Yaskawa INFORM job: SKRZYNIA_5440_0_STOPNI_2OBR.JBI

/JOB
//NAME SKRZYNIA_5440_0_STOPNI_2OBR
///FOLDERNAME 02-SKRZYNIE_JOBS
//POS
///NPOS 734,734,0,54,0,0
///TOOL 0
///POSTYPE PULSE
///PULSE
C00000=1055,-24125,84372,288,19725,204
C00001=0,-15438,65714,0,-68532,0
C00002=4718,-16587,59952,3396,-65485,-935
C00003=32997,-21499,42555,27623,-61436,21376
C00004=31759,-20688,42932,26837,-60850,21559
C00005=28987,-21156,42712,24818,-60442,22222
C00006=33447,-21964,42352,27886,-61721,21330
C00007=37687,-23357,41794,30651,-63289,20620
C00008=38979,-19018,48057,32961,-64962,20678
C00009=37261,-18075,48526,31902,-64209,20901
C00010=35830,-17198,48994,31015,-63571,21092
C00011=34080,-17614,48768,29780,-63290,21485
C00012=37261,-18075,48526,31902,-64209,20901
C00013=47373,-21912,40596,41149,-66086,26950
C00014=4718,-16587,59952,3396,-65485,-935
C00015=32997,-21499,42555,27623,-61436,21376
C00016=31759,-20688,42932,26837,-60850,21559
C00017=28987,-21156,42712,24818,-60442,22222
C00018=33447,-21964,42352,27886,-61721,21330
C00019=37687,-23357,41794,30651,-63289,20620
C00020=38979,-19018,48057,32961,-64962,20678
C00021=37261,-18075,48526,31902,-64209,20901
C00022=35830,-17198,48994,31015,-63571,21092
C00023=34080,-17614,48768,29780,-63290,21485
C00024=37261,-18075,48526,31902,-64209,20901
C00025=47373,-21912,40596,41149,-66086,26950
C00026=45033,-20851,41104,39798,-65001,27223
C00027=42790,-19693,41704,38494,-63946,27495
C00028=41070,-20182,41442,37324,-63566,27891
C00029=45033,-20851,41104,39798,-65001,27223
C00030=45033,-20851,41104,39798,-65001,27223
C00031=59624,-29540,14278,64846,-60867,16042
C00032=57357,-28542,14780,63940,-59509,16120
C00033=56188,-29140,14476,63237,-58995,16387
C00034=59588,-29370,14363,64862,-60819,16012
C00035=62924,-29779,15793,65870,-63073,16252
C00036=59724,-28781,16276,64511,-61238,16415
C00037=57764,-27936,16704,63709,-60078,16488
C00038=56408,-28589,16373,62897,-59486,16787
C00039=59724,-28781,16276,64511,-61238,16415
C00040=59800,-47064,-28857,95901,-51687,-331
C00041=35771,-53551,-30995,85975,-27014,914
C00042=34295,-52413,-30674,86854,-26051,280
C00043=32024,-52970,-30833,85668,-24589,638
C00044=35771,-53551,-30995,85975,-27014,914
C00045=87562,-48087,-13810,78020,-75252,11220
C00046=10104,-46603,4759,11228,-37390,-5046
C00047=0,-52280,40443,0,6876,0
C00048=1529,-42140,58025,-5964,2417,3265
C00049=49472,-39353,6917,53118,-50908,20251
C00050=45058,-39356,3832,51653,-47640,20099
C00051=42883,-38319,4163,50577,-46309,20295
C00052=40255,-38926,3967,48502,-45334,21060
C00053=46774,-39679,3737,52663,-48537,19827
C00054=48708,-40455,3517,53615,-49689,19657
C00055=43798,-39237,3871,50850,-47027,20335
C00056=41951,-38324,4161,49930,-45891,20507
C00057=39836,-38844,3994,48234,-45126,21137
C00058=48489,-40338,3551,53521,-49551,19665
C00059=48489,-40338,3551,53521,-49551,19665
C00060=44432,-39026,3936,51363,-47247,20139
C00061=42487,-38069,4248,50403,-46050,20315
C00062=39061,-38795,4009,47695,-44769,21310
C00063=44432,-39026,3936,51363,-47247,20139
C00064=57930,-43229,1921,58550,-54632,18533
C00065=40247,-55452,-40505,109199,-33003,-7808
C00066=33946,-52082,-43455,125156,-33578,-16149
C00067=32704,-50650,-42908,126591,-33384,-17037
C00068=30549,-51326,-43170,127422,-32071,-17630
C00069=37275,-55997,-51641,126340,-37028,-16651
C00070=64697,-70559,-57820,113226,-48939,-6101
C00071=1817,-44984,2816,-3462,-45659,1296
C00072=1148,-56354,34370,-22,3827,-10
C00073=0,-52280,40443,0,6876,0
C00074=0,-49898,44897,0,-65513,0
C00075=48645,-40151,10421,50724,-47615,19638
C00076=35184,-37395,11059,41539,-41116,22069
C00077=33403,-36378,11356,40435,-40041,22314
C00078=30649,-36829,11220,37805,-39247,23256
C00079=35184,-37395,11059,41539,-41116,22069
C00080=36291,-43239,-398,48566,-36532,18743
C00081=34674,-42363,-182,47694,-35492,18907
C00082=33151,-41445,67,46884,-34487,19058
C00083=30501,-41913,-62,44164,-33547,20068
C00084=34674,-42363,-182,47694,-35492,18907
C00085=54016,-42729,8218,55932,-50472,20462
C00086=-31499,-58302,-23356,15027,12889,-13082
C00087=-52768,-43016,-26078,18373,38595,-18774
C00088=-89470,-32103,-32973,29905,69139,-31512
C00089=-68838,-26884,-24872,16972,64732,-23076
C00090=-53036,-11528,-12218,12363,64665,-17409
C00091=-51536,-9474,-10276,11905,64649,-16876
C00092=-51739,-9114,-7787,12104,63269,-17104
C00093=-53036,-11528,-12218,12363,64665,-17409
C00094=-17541,-26226,-24397,927,59032,-5038
C00095=-17541,-26226,-24397,927,59032,-5038
C00096=-16950,-23991,-22741,715,59568,-4818
C00097=-17036,-23563,-20101,755,58071,-4857
C00098=-17541,-26226,-24397,927,59032,-5038
C00099=34102,-23192,-21614,-15638,64271,13209
C00100=33423,-21885,-20599,-15423,64418,12942
C00101=32426,-19856,-18975,-15106,64629,12551
C00102=32578,-19611,-17013,-15290,63535,12762
C00103=33423,-21885,-20599,-15423,64418,12942
C00104=59339,-6070,-6417,-20979,72191,20891
C00105=59339,-6070,-6417,-20979,72191,20891
C00106=57897,-4256,-4562,-20702,71913,20431
C00107=58108,-3992,-2506,-20878,70835,20713
C00108=59339,-6070,-6417,-20979,72191,20891
C00109=42744,-35904,-30225,-18322,62562,16651
C00110=-53036,-11528,-12218,12363,64665,-17409
C00111=-77982,-26538,-29134,27151,66629,-27745
C00112=-70983,-8594,-1966,26503,59809,-49670
C00113=-80152,19776,40785,37351,72704,-50428
C00114=-79984,20154,42529,37516,71911,-50638
C00115=-79233,18397,40079,37458,71885,-50340
C00116=-79984,20154,42529,37516,71911,-50638
C00117=-73519,23289,38838,28890,77081,-45618
C00118=-73519,24511,42682,29072,75582,-46027
C00119=-73519,23289,38838,28890,77081,-45618
C00120=-88897,15706,42282,50101,71325,-56974
C00121=-88897,15706,42282,50101,71325,-56974
C00122=-87612,12343,37838,50071,70996,-56519
C00123=-85283,14202,40272,50301,69633,-56165
C00124=-87338,12550,38107,50098,70839,-56476
C00125=-84952,-1789,13569,34660,47724,-58955
C00126=-67641,-1674,11109,10330,44856,-44725
C00127=-66443,961,13975,9688,44721,-44210
C00128=-67641,-1674,11109,10330,44856,-44725
C00129=-67641,-376,15347,10694,42950,-44967
C00130=-67641,-1674,11109,10330,44856,-44725
C00131=-79040,417,20398,15965,28992,-57786
C00132=-76655,5212,30978,15501,25024,-57306
C00133=-76655,6949,35816,16758,23084,-57955
C00134=-76655,5212,30978,15501,25024,-57306
C00135=-74761,6919,33010,13466,24593,-56049
C00136=-80460,-2874,12270,15804,32253,-57809
C00137=-61258,-29124,-13156,26560,43617,-22150
C00138=-30420,-40507,-29240,27153,53235,15188
C00139=-18589,-38725,-21450,23338,47896,18931
C00140=-17722,-35233,-16455,23322,46926,19051
C00141=-17722,-33749,-12435,23948,45421,18620
C00142=-17722,-33892,-12819,23887,45564,18661
C00143=-16677,-31133,-11209,23138,46167,19311
C00144=-17819,-35820,-17540,23246,47228,19090
C00145=-74104,-11494,-6266,31916,75042,4269
C00146=-71226,-7329,2631,32115,71468,4273
C00147=-71226,-6504,5446,32343,70365,3922
C00148=-71226,-6611,5086,32313,70505,3967
C00149=-68386,-4058,7675,32040,69573,4789
C00150=-73314,-9412,-353,32206,72648,3829
C00151=51751,-31069,-22965,-10739,49070,48663
C00152=49028,-23852,-11575,-9841,46366,47823
C00153=49028,-23004,-8935,-10039,45204,47956
C00154=49028,-23118,-9286,-10013,45357,47939
C00155=47000,-20813,-7527,-8928,45644,47024
C00156=50476,-26208,-15307,-10408,47325,48332
C00157=90602,-5375,6902,-38786,69848,59444
C00158=83174,19950,50269,-44999,67580,58220
C00159=82362,17902,47383,-44926,67511,57879
C00160=83515,19072,48341,-44798,68200,58056
C00161=78091,19382,40247,-36371,72286,52960
C00162=78091,20664,44011,-36670,70997,53443
C00163=78091,19382,40247,-36371,72286,52960
C00164=88699,7296,38566,-55615,63182,60372
C00165=86803,3068,32674,-55410,62638,59657
C00166=84852,4315,34115,-55564,61561,59330
C00167=86803,3068,32674,-55410,62638,59657
C00168=92770,-2803,21719,-53893,67577,59421
C00169=73393,-10627,10934,-27897,30744,62458
C00170=70789,-6606,18800,-27824,27830,62140
C00171=69654,-4593,20814,-26755,27596,61444
C00172=70789,-6606,18800,-27824,27830,62140
C00173=70789,-5070,23059,-29482,26284,63017
C00174=70789,-6606,18800,-27824,27830,62140
C00175=83486,-8736,6503,-27040,35338,66550
C00176=77831,-2041,26192,-25270,18452,68895
C00177=77967,1961,32070,-26860,17569,69698
C00178=77967,5243,40752,-32914,14549,72656
C00179=77967,1961,32070,-26860,17569,69698
C00180=74560,4730,35257,-21622,16551,66717
C00181=77967,1961,32070,-26860,17569,69698
C00182=81109,-22356,2664,-22493,33121,60116
C00183=86168,-49730,-13668,-23926,46819,49343
C00184=44183,-52048,-7537,-24795,46064,51426
C00185=0,-52280,40443,0,6876,0
C00186=0,-52280,40443,0,6876,0
C00187=33629,-57276,-6399,46271,-24969,-2804
C00188=75493,-63502,-64712,103874,-64610,-6298
C00189=47506,-58574,-62752,109785,-45896,-10707
C00190=43794,-60202,-65944,114374,-43231,-9322
C00191=55379,-67378,-68041,108237,-48773,-4935
C00192=62671,-64213,-64640,104431,-56093,-7372
C00193=28458,-50318,6850,47420,-25887,-3347
C00194=0,-52280,40443,0,6876,0
C00195=1055,-24125,84372,288,19725,204
C00196=0,-15438,65714,0,-68532,0
C00197=0,-15438,65714,966,-70097,42926
C00198=69988,-9219,57065,61610,-82752,27767
C00199=63113,-6157,59685,58080,-79692,28271
C00200=46309,-5455,68070,40267,-75151,29719
C00201=49471,-5188,67710,43421,-76082,29577
C00202=63113,-6157,59685,58080,-79692,28271
C00203=69988,-9219,57065,61610,-82752,27767
C00204=0,-15438,65714,966,-70097,42926
C00205=0,-15438,65714,0,-68532,0
C00206=1055,-24125,84372,288,19725,204
C00207=1055,-24125,84372,288,19725,204
C00208=0,-41971,13909,0,6774,1
C00209=-55064,-17017,13106,20113,45767,-35735
C00210=-85641,-3161,12660,31281,67420,-55579
C00211=-77611,9747,38455,32702,57795,-55547
C00212=-77611,9747,38455,32702,57795,-55547
C00213=-80481,23547,61641,37204,60115,-56891
C00214=-80479,11681,28780,33754,71138,-52780
C00215=-73572,15026,34389,33675,67405,-51294
C00216=-73572,20195,49236,35290,62248,-53161
C00217=-82806,26311,53816,38180,73291,-53604
C00218=-71695,3747,16001,30713,64750,-51022
C00219=-70421,5575,20105,30867,63066,-51036
C00220=-35543,-20105,-5144,22821,50284,-40173
C00221=-37830,-23193,-8618,23571,50957,-40982
C00222=11136,-28839,-12562,1025,41780,-20887
C00223=20486,-27077,-7346,-12554,38415,-10736
C00224=59545,-9921,5571,-27063,51925,3267
C00225=55110,-17412,-5825,-19778,50988,-2825
C00226=79390,11759,28162,-35512,71262,52960
C00227=74811,13878,33986,-35807,67493,52464
C00228=74942,18762,48004,-37392,62815,54352
C00229=76815,18630,46530,-37158,64288,54543
C00230=79390,11759,28162,-35512,71262,52960
C00231=10831,-54278,-29128,-6468,39852,-5090
C00232=-67200,-10549,24402,-3189,24913,-39001
C00233=-75122,-2194,12822,3152,39225,-43427
C00234=-77516,10189,32861,8493,33365,-45533
C00235=-75154,17575,49272,7885,27457,-44928
C00236=-68113,9932,38901,1157,28472,-40453
C00237=-67114,5383,31515,9208,32648,-43213
C00238=-66450,3998,29285,10896,33890,-43630
C00239=-66374,3101,28136,14657,35566,-44954
C00240=-66576,452,24763,27028,43375,-49112
C00241=-69928,4230,30673,35488,50431,-52676
C00242=-77050,-3138,8526,33226,61087,-51698
C00243=-67200,-10549,24402,-3189,24913,-39001
C00244=0,-52280,40443,83103,28146,-16510
C00245=99993,-20782,22705,-13349,24734,56519
C00246=67200,-10549,24402,3189,24913,39001
C00247=75122,-2194,12822,-3152,39225,43427
C00248=74323,5203,27259,-5972,33194,43789
C00249=74015,16414,48063,-6821,27325,44224
C00250=56519,1138,28747,9235,29393,33453
C00251=55467,619,28251,10155,29461,32830
C00252=56374,-724,25854,4078,30541,35419
C00253=56480,-7201,15910,-17697,38451,43334
C00254=68252,956,25699,-34035,49810,51639
C00255=77050,-3138,8526,-33226,61087,51698
C00256=67200,-10549,24402,3189,24913,39001
C00257=0,-52280,40443,-83103,28146,16510
C00258=-99993,-20782,22705,13349,24734,-56519
C00259=-91125,453,39555,30378,52425,-51131
C00260=-81425,-5449,14825,37552,56592,-47667
C00261=-81425,-10835,-2515,34915,62871,-45127
C00262=-79239,4305,16082,37593,68846,-50182
C00263=-81302,5892,27588,46359,62943,-54679
C00264=-82227,19402,59913,51524,57300,-60581
C00265=-84844,8890,27031,38640,69740,-53449
C00266=-90096,4679,14083,37467,76581,-51973
C00267=-87885,29238,52923,40761,81198,69685
C00268=-84355,23847,39024,40698,83720,72224
C00269=-81960,27335,46957,41070,80536,71891
C00270=-82643,24718,50492,48951,72637,70260
C00271=-90480,18737,31939,47254,81986,71631
C00272=-94217,10634,17426,46901,86469,-59967
C00273=-81425,-10835,-2515,34915,62871,-45127
C00274=-81425,-5449,14825,37552,56592,-47667
C00275=-94290,-610,44819,32366,49686,-53459
C00276=0,-55136,17047,60468,32096,-4233
C00277=99993,-20782,22705,-13349,24734,56519
C00278=91125,453,39555,-30378,52425,51131
C00279=81425,-5449,14825,-37552,56592,47667
C00280=81425,-10835,-2515,-34915,62871,45127
C00281=79239,4305,16082,-37593,68846,50182
C00282=83239,4964,30263,-50637,62037,57149
C00283=83991,16425,61235,-57769,55250,63273
C00284=93928,7973,40920,-53095,64494,61640
C00285=75109,22299,39152,-26915,78743,47998
C00286=79256,17348,34699,-33448,76412,88212
C00287=79932,23608,50901,-39863,71219,88955
C00288=76220,30771,63034,-41386,67395,88927
C00289=86322,16060,37848,-39554,76452,89287
C00290=87424,-1569,9538,-38190,72401,52253
C00291=81425,-10835,-2515,-34915,62871,45127
C00292=92850,-11266,9233,-39092,60986,50964
C00293=28366,-40369,19479,-5635,23506,17663
C00294=-80334,-19501,31260,21216,42469,-40219
C00295=-80621,-32280,-9061,25825,59412,-41877
C00296=-80621,-37319,-22868,24573,64555,-40576
C00297=-75108,-2453,16462,35304,60348,-42510
C00298=-72231,7240,33473,36511,55681,-43130
C00299=-35770,-19109,7486,28512,40799,-31761
C00300=-39606,-22901,-1163,28356,44724,-32188
C00301=15344,-29112,-5358,-2858,33820,-6852
C00302=13390,-24012,2637,-1527,32105,-7853
C00303=57983,-8601,15571,-27088,42703,12849
C00304=60973,-17187,4937,-27817,44388,13718
C00305=60973,-17187,4937,-27817,44388,13718
C00306=-13287,-42463,-12044,19170,31021,-23010
C00307=-17374,-21287,20534,22794,29118,-26096
C00308=13276,-20759,18622,-1911,29377,-7028
C00309=39924,-14247,19329,-14795,35999,4396
C00310=41528,-14133,18797,-15449,36702,5040
C00311=57001,-5890,26499,-21893,40771,11494
C00312=64054,-19541,3059,-29141,44956,15011
C00313=51466,-33957,-1499,-46586,51805,23434
C00314=17032,-20770,22044,-28854,30468,11088
C00315=-9868,-18638,14971,-8492,38486,-5199
C00316=-40562,-13194,19800,9508,35447,-20184
C00317=-41848,-12620,20103,10165,35810,-20773
C00318=-57278,-4046,28217,17578,39066,-27653
C00319=-71680,-19835,10874,33863,39440,-36917
C00320=-20806,-37586,-12792,9951,42782,-18031
C00321=29087,-45372,27330,-13325,19529,9021
C00322=0,-52280,40443,0,6876,0
C00323=0,-52280,40443,0,6876,0
C00324=0,-17525,61946,0,273,32004
C00325=54446,-4421,37881,-48560,57645,57448
C00326=45059,-5790,38757,-53071,45868,54447
C00327=54214,-14697,41967,-94765,49928,76221
C00328=38139,-25233,26108,-101870,33233,74060
C00329=36109,-19033,24738,-65594,32215,56497
C00330=50018,-7105,51930,-74419,40156,68238
C00331=45059,-5790,38757,-53071,45868,54447
C00332=0,-17525,61946,0,273,32004
C00333=0,-52280,40443,0,6876,0
C00334=0,-52280,40443,0,6876,0
C00335=0,-52280,40443,0,6876,0
C00336=0,-52280,40443,0,-42737,40640
C00337=0,-52280,40443,0,-42737,40640
C00338=64551,-35409,28076,75550,-44539,17239
C00339=49799,-25338,45366,61341,-39751,21495
C00340=45731,-22710,35392,68644,-36821,18294
C00341=24330,-29244,24695,37362,-28659,27524
C00342=19913,-27131,30534,27440,-28693,31340
C00343=43117,-27612,29118,67655,-35359,18183
C00344=39863,-22026,47404,54615,-35502,22403
C00345=0,-52277,40442,0,6872,2
C00346=0,-38538,66749,0,-898,0
C00347=0,-52280,40443,0,-79033,35417
C00348=46775,-35113,22190,42926,-67531,20697
C00349=52587,-26056,25345,47610,-66542,17970
C00350=46026,-25515,24478,44186,-63240,18818
C00351=46112,-27744,19536,44836,-62075,18165
C00352=53914,-29436,22058,48262,-67266,17843
C00353=63113,-6157,59685,58080,-79692,28271
C00354=46665,-5556,67979,40480,-75262,29672
C00355=49442,-5188,67743,43340,-76070,29564
C00356=58009,-5921,62835,52447,-77983,28714
C00357=58009,-5921,62835,52447,-77983,28714
C00358=53914,-29436,22058,48262,-67266,17843
C00359=46775,-35113,22190,42926,-67531,20697
C00360=77624,-37863,9189,71219,-67328,18688
C00361=32759,-44624,-7410,48391,-34222,22497
C00362=27557,-32134,11789,69915,-21290,13317
C00363=40062,-38096,12902,49436,-40427,24267
C00364=0,-52280,40443,0,-61239,28081
C00365=404,-42897,57020,-1574,2523,869
C00366=0,-52280,40443,0,6876,0
C00367=-99253,-13690,44082,59847,13407,-31313
C00368=-87814,-12734,20141,45739,-14352,-64418
C00369=-86556,-6739,30659,41315,-16837,-62092
C00370=-85114,-6068,31313,43868,-17408,-63130
C00371=-86280,-6613,30781,41818,-16944,-62296
C00372=-86999,-5595,31777,40735,-16589,-61870
C00373=-86280,-6613,30781,41818,-16944,-62296
C00374=-90751,-10996,-2268,-12017,29723,-39494
C00375=-90751,-10996,-2268,-12017,29723,-39494
C00376=-90751,-9656,2306,-12858,27632,-39044
C00377=-90751,-10996,-2268,-12017,29723,-39494
C00378=-86125,-12470,22545,29004,-25567,-58412
C00379=-83883,-11340,22525,32952,-25567,-60136
C00380=-82768,-10824,22986,34487,-25904,-60776
C00381=-83883,-11340,22525,32952,-25567,-60136
C00382=-85143,-9772,23941,31487,-24966,-59556
C00383=-83883,-11340,22525,32952,-25567,-60136
C00384=-85732,-21202,11427,30682,-24763,-59235
C00385=-84150,-10929,23786,31981,-25941,-59678
C00386=-83036,-10419,24246,33504,-26268,-60308
C00387=-84150,-10929,23786,31981,-25941,-59678
C00388=-85291,-9507,25078,30650,-25411,-59154
C00389=-84150,-10929,23786,31981,-25941,-59678
C00390=-85786,-16909,14677,31743,-23900,-59790
C00391=-84150,-10498,24888,31517,-26306,-59436
C00392=-83174,-10052,25293,32841,-26587,-59984
C00393=-84150,-10498,24888,31517,-26306,-59436
C00394=-85258,-9112,26156,30226,-25800,-58928
C00395=-84150,-10498,24888,31517,-26306,-59436
C00396=-87841,-18519,13420,28367,-23534,-58339
C00397=-84150,-10465,24972,31484,-26336,-59417
C00398=-83241,-10052,25348,32714,-26598,-59924
C00399=-84150,-10465,24972,31484,-26336,-59417
C00400=-85145,-9228,26102,30329,-25881,-58963
C00401=-84150,-10465,24972,31484,-26336,-59417
C00402=-86371,-18277,13606,30568,-23951,-59265
C00403=-84345,-11688,21985,32461,-25312,-59957
C00404=-83211,-11173,22442,34044,-25650,-60618
C00405=-84345,-11688,21985,32461,-25312,-59957
C00406=-85283,-10526,23025,31366,-24861,-59525
C00407=-84345,-11688,21985,32461,-25312,-59957
C00408=-86191,-19647,12567,30467,-24278,-59187
C00409=-84345,-10877,24073,31552,-26006,-59481
C00410=-83051,-10286,24607,33321,-26381,-60213
C00411=-84345,-10877,24073,31552,-26006,-59481
C00412=-85179,-9842,25009,30582,-25619,-59100
C00413=-84345,-10877,24073,31552,-26006,-59481
C00414=-85438,-18022,14839,31140,-24818,-59429
C00415=-84247,-11820,22550,32049,-25753,-59727
C00416=-84104,-10976,23642,32111,-25899,-59738
C00417=-82990,-10465,24105,33639,-26227,-60372
C00418=-84104,-10976,23642,32111,-25899,-59738
C00419=-84898,-9998,24525,31196,-25529,-59378
C00420=-84104,-10976,23642,32111,-25899,-59738
C00421=-86610,-16845,14732,30573,-23614,-59301
C00422=-84104,-10864,23927,31990,-25993,-59674
C00423=-82824,-10273,24459,33737,-26370,-60397
C00424=-84104,-10864,23927,31990,-25993,-59674
C00425=-84789,-10021,24690,31200,-25673,-59363
C00426=-84104,-10864,23927,31990,-25993,-59674
C00427=-83806,-19585,12613,33764,-25080,-60559
C00428=-83924,-10205,25475,31619,-26533,-59453
C00429=-82780,-9675,25960,33156,-26866,-60087
C00430=-83924,-10205,25475,31619,-26533,-59453
C00431=-84478,-9530,26093,30986,-26280,-59206
C00432=-83924,-10205,25475,31619,-26533,-59453
C00433=-87149,-17993,13826,29513,-23647,-58830
C00434=-84920,-13182,20975,31162,-25481,-59361
C00435=-83711,-10572,24852,32056,-26475,-59649
C00436=-82779,-10142,25241,33309,-26748,-60166
C00437=-83711,-10572,24852,32056,-26475,-59649
C00438=-84370,-9774,25579,31305,-26170,-59356
C00439=-83711,-10572,24852,32056,-26475,-59649
C00440=-83642,-3679,42021,23358,-36761,-56118
C00441=-85886,-5975,41264,18964,-40261,-54782
C00442=-83919,-11632,22322,32811,-25616,-60079
C00443=-82884,-11162,22742,34234,-25925,-60671
C00444=-83919,-11632,22322,32811,-25616,-60079
C00445=-84723,-10654,23196,31887,-25230,-59715
C00446=-83919,-11632,22322,32811,-25616,-60079
C00447=-87348,-16035,7353,17528,-35245,-56477
C00448=-86244,-15062,8172,18754,-35315,-57058
C00449=-86244,-16649,3638,19674,-33501,-57585
C00450=-85308,-16228,3988,20718,-33648,-58082
C00451=-86244,-16649,3638,19674,-33501,-57585
C00452=-86740,-15973,4201,19194,-33277,-57362
C00453=-86244,-16649,3638,19674,-33501,-57585
C00454=-73780,-8639,20128,34258,-51705,-52097
C00455=-90711,-17528,-28778,11328,-28245,-57111
C00456=-92565,-19610,-33223,7138,-24591,-57051
C00457=-91512,-19116,-32812,8551,-24603,-57834
C00458=-92565,-19610,-33223,7138,-24591,-57051
C00459=-93003,-18716,-32476,6600,-24397,-56752
C00460=-92565,-19610,-33223,7138,-24591,-57051
C00461=-92565,-19610,-33223,7138,-24591,-57051
C00462=-95836,-54375,-51122,6031,-17685,-48210
C00463=-95836,-54375,-51122,6031,-17685,-48210
C00464=-43821,-47238,-2775,-3022,56549,-3681
C00465=-20126,-26882,59542,2406,16879,-9162
C00466=-20126,-26882,59542,2406,16879,-9162
C00467=98601,-10520,92678,4674,-40855,-9615
C00468=95537,-19831,-2695,-2933,-44471,35837
C00469=92548,-20391,-28429,-6186,-30623,55200
C00470=91429,-17018,-28974,-8057,-27827,56250
C00471=91429,-17018,-28974,-8057,-27827,56250
C00472=90371,-16495,-28521,-9286,-27856,56953
C00473=91429,-17018,-28974,-8057,-27827,56250
C00474=92033,-15799,-27911,-7415,-27588,55880
C00475=91429,-17018,-28974,-8057,-27827,56250
C00476=92548,-20391,-28429,-6186,-30623,55200
C00477=91156,-15018,-4648,-8036,-38181,54813
C00478=90585,-14766,-4428,-8565,-38201,55100
C00479=88830,-13959,-3717,-10186,-38284,55977
C00480=89897,-14456,-4157,-9202,-38230,55445
C00481=90761,-12944,-2809,-8452,-37927,55043
C00482=89897,-14456,-4157,-9202,-38230,55445
C00483=89910,-11217,67535,-9455,-58896,55399
C00484=89910,-11217,67535,-9455,-58896,55399
C00485=85786,-16735,14816,-31782,-23869,59812
C00486=83514,-12996,17929,-35760,-24132,61552
C00487=82251,-12406,18443,-37550,-24551,62308
C00488=83514,-12996,17929,-35760,-24132,61552
C00489=84258,-12095,18717,-34917,-23742,61217
C00490=83514,-12996,17929,-35760,-24132,61552
C00491=87149,-17993,13826,-29513,-23647,58830
C00492=83118,-12818,18089,-36330,-24263,61791
C00493=81915,-12248,18589,-38020,-24666,62504
C00494=83118,-12818,18089,-36330,-24263,61791
C00495=83897,-11882,18912,-35460,-23856,61445
C00496=83118,-12818,18089,-36330,-24263,61791
C00497=83806,-19585,12613,-33764,-25080,60559
C00498=82998,-13006,17925,-36445,-24332,61826
C00499=81675,-12378,18472,-38297,-24777,62607
C00500=82998,-13006,17925,-36445,-24332,61826
C00501=83876,-11958,18841,-35466,-23874,61442
C00502=82998,-13006,17925,-36445,-24332,61826
C00503=86610,-16845,14732,-30573,-23614,59301
C00504=82493,-13239,17725,-37070,-24559,62089
C00505=81406,-12724,18174,-38578,-24928,62723
C00506=82493,-13239,17725,-37070,-24559,62089
C00507=83436,-12134,18690,-36041,-24064,61684
C00508=82493,-13239,17725,-37070,-24559,62089
C00509=84814,-16043,15376,-33312,-24093,60464
C00510=82555,-13613,17404,-36910,-24580,62015
C00511=81384,-13062,17878,-38534,-24974,62698
C00512=82555,-13613,17404,-36910,-24580,62015
C00513=83566,-12434,18427,-35805,-24047,61580
C00514=82555,-13613,17404,-36910,-24580,62015
C00515=86191,-19647,12567,-30467,-24278,59187
C00516=82500,-13648,17375,-36975,-24607,62039
C00517=81467,-13161,17792,-38413,-24955,62645
C00518=82500,-13648,17375,-36975,-24607,62039
C00519=83481,-12505,18364,-35905,-24087,61617
C00520=82500,-13648,17375,-36975,-24607,62039
C00521=86371,-18277,13606,-30568,-23951,59265
C00522=82904,-13790,17251,-36416,-24470,61808
C00523=81715,-13237,17726,-38081,-24865,62509
C00524=82904,-13790,17251,-36416,-24470,61808
C00525=83686,-12878,18037,-35556,-24055,61469
C00526=82904,-13790,17251,-36416,-24470,61808
C00527=87841,-18519,13420,-28367,-23534,58339
C00528=82748,-13879,17174,-36603,-24542,61883
C00529=81692,-13388,17594,-38077,-24893,62505
C00530=82748,-13879,17174,-36603,-24542,61883
C00531=83607,-12881,18032,-35663,-24082,61515
C00532=82748,-13879,17174,-36603,-24542,61883
C00533=85786,-16909,14677,-31743,-23900,59790
C00534=82520,-14198,16902,-36833,-24674,61972
C00535=81460,-13708,17319,-38301,-25026,62591
C00536=82520,-14198,16902,-36833,-24674,61972
C00537=83571,-12989,17938,-35691,-24113,61524
C00538=82520,-14198,16902,-36833,-24674,61972
C00539=85732,-21202,11427,-30682,-24763,59235
C00540=82398,-14365,16763,-36952,-24745,62014
C00541=81172,-13798,17245,-38643,-25153,62725
C00542=82398,-14365,16763,-36952,-24745,62014
C00543=83600,-12984,17944,-35650,-24102,61504
C00544=82398,-14365,16763,-36952,-24745,62014
C00545=92346,-18713,13565,-21110,-22545,55257
C00546=82794,-13980,17083,-36511,-24538,61844
C00547=81518,-13384,17592,-38292,-24965,62594
C00548=82794,-13980,17083,-36511,-24538,61844
C00549=83714,-12912,18003,-35501,-24048,61445
C00550=82794,-13980,17083,-36511,-24538,61844
C00551=86140,-12802,12665,-93523,-10743,85795
C00552=86140,-12802,12665,-93523,-10743,85795
C00553=85030,-12289,13120,-93723,-11463,85776
C00554=86140,-12802,12665,-93523,-10743,85795
C00555=86958,-11660,13681,-94506,-10238,86349
C00556=85239,-16743,-4327,42764,21357,45785
C00557=86630,-1784,19103,24023,25413,52215
C00558=86630,-582,22633,25405,24035,51499
C00559=86630,-2021,18396,23764,25694,52349
C00560=83866,-23485,-9665,46715,21048,43706
C00561=73745,-37787,-30345,49345,28485,41761
C00562=85045,-36869,-4353,-28502,-22832,52282
C00563=0,-24029,84339,0,19981,0
C00564=0,-24029,84339,0,19981,0
C00565=3172,-24246,80980,3465,15913,689
C00566=-86563,-26985,13879,10257,-21548,-45530
C00567=-86191,-19647,12567,30467,-24278,-59187
C00568=-83221,-13587,17636,37793,-25116,-62228
C00569=-92023,-13764,14621,12306,-18616,-51487
C00570=-95023,-13777,14330,1211,-18003,-46636
C00571=-84074,-17488,11256,38660,-23649,-62784
C00572=-73679,-33270,1000,44272,-31600,-64253
C00573=-86926,-60758,23267,6576,1160,-9545
C00574=0,-52280,40443,0,6876,0
C00575=82475,-58079,26734,835,4084,4444
C00576=97932,-26840,7691,8784,-23444,42538
C00577=87166,-16607,16322,-25365,-24201,56345
C00578=84825,-11409,21703,-28959,-24702,57870
C00579=84878,-11056,22701,-28451,-25053,57612
C00580=85100,-26994,10417,-24982,-28140,55821
C00581=0,-52280,40443,0,6876,0
C00582=0,-52280,40443,0,6876,0
C00583=-90140,-60305,18108,-2708,1721,-7625
C00584=-95594,-27428,6866,-4663,-19832,-42154
C00585=-98688,-13767,16447,-18366,-10080,-35766
C00586=-98964,-4977,31041,-27811,-8682,-30400
C00587=-98916,-3735,32751,-30964,-8053,-28728
C00588=-99892,-12729,3741,-149109,-12188,27676
C00589=-96569,-4256,22865,-166316,-8784,33175
C00590=-98555,-11355,6708,-165016,-14703,32370
C00591=-99753,-15088,-24382,-164889,-47912,36555
C00592=-96569,-4256,22865,-166316,-8784,33175
C00593=-97622,-14456,11637,-152676,-5975,26484
C00594=-90140,-60305,18108,-2708,1721,-7625
C00595=0,-52280,40443,0,6876,0
C00596=84259,-57935,27522,-3761,3673,6310
C00597=86507,-39672,4297,-27618,-16640,46340
C00598=73669,-37119,-20783,-92053,-19719,85232
C00599=86539,-20830,1725,-71850,-11773,76853
C00600=94927,-16191,10904,-46169,-1414,61414
C00601=97577,-11989,12425,-54085,4211,65686
C00602=97819,-13198,9149,-43063,5201,60524
C00603=98855,-10677,214,-11203,24557,44562
C00604=98625,785,31085,-10261,24068,43352
C00605=97715,6871,36042,-10941,32148,42233
C00606=98966,17478,50100,-9488,29710,42739
C00607=100487,-9453,-1206,-10413,41328,41147
C00608=96250,-19428,-8283,-4838,27297,37910
C00609=86507,-39672,4297,-27618,-16640,46340
C00610=84259,-57935,27522,-3761,3673,6310
C00611=0,-52280,40443,0,6876,0
C00612=0,-27933,77061,0,20812,0
C00613=0,-27933,77061,0,20812,0
C00614=0,-52280,40443,0,6876,0
C00615=-91970,-60791,14435,-3343,512,-9412
C00616=-98647,-24138,10005,-11519,-21203,-39749
C00617=-99883,-13980,22886,-11640,-25090,-40341
C00618=-99702,-9154,61728,-1148,-61809,-40243
C00619=-84328,-13042,29707,23458,-33731,-54641
C00620=-83186,-4072,39316,25807,-34757,-55633
C00621=-82903,-4302,38720,26369,-34472,-55857
C00622=-76259,-18287,26646,31659,-38322,-57579
C00623=-89741,-28009,12101,4461,-28076,-46404
C00624=-91970,-60791,14435,-3343,512,-9412
C00625=0,-52280,40443,0,6876,0
C00626=91083,-60784,14823,-9043,-825,15173
C00627=83869,-19403,12921,-33769,-24740,60260
C00628=83869,-19403,12921,-33769,-24740,60260
C00629=83932,-19538,53415,-33663,-71112,60249
C00630=83932,-19538,53415,-33663,-71112,60249
C00631=82480,-12247,21118,-35440,-26416,60009
C00632=82280,-11332,19892,-37560,-25279,61090
C00633=81927,-9347,24735,-35767,-26869,60100
C00634=79790,-20261,14917,-36681,-28829,60258
C00635=76554,-29711,-1870,-46042,-25952,65654
C00636=91083,-60784,14823,-9043,-825,15173
C00637=0,-52280,40443,0,6876,0
C00638=-91526,-60598,16699,7584,176,-13289
C00639=-81382,-25890,9219,35455,-25500,-59095
C00640=-86453,-20958,12525,30076,-22568,-57089
C00641=-86589,-16097,16237,31250,-21582,-57704
C00642=-98933,-11298,20505,-13970,-18736,-37953
C00643=-98403,-10946,21278,-11768,-18626,-39241
C00644=-89939,-20003,13253,27082,-21802,-55813
C00645=-85529,-37325,-10065,38133,-20822,-60794
C00646=-81326,-27507,8265,35533,-26282,-59001
C00647=-91415,-60262,16631,7870,-73,-13734
C00648=24,-24029,84339,7,19981,5
C00649=100404,-52373,45687,-1822,14816,-5144
C00650=75939,-26469,7919,-40869,-29645,63133
C00651=81882,-22565,10470,-35355,-26404,61107
C00652=82801,-12246,21732,-34208,-26055,60642
C00653=91931,-10448,23719,-8474,-22170,49733
C00654=96901,-9497,26324,6381,-23158,43441
C00655=77262,-23244,14300,-38922,-31295,61912
C00656=78410,-22868,15324,-38001,-30064,61274
C00657=96357,-33562,33410,58602,-23427,10353
C00658=568,-24029,84339,168,19981,112
C00659=-91970,-60791,14435,-3343,512,-9412
C00660=-98991,-22833,11519,-12824,-17638,-36336
C00661=-86376,-13627,18436,38326,-18406,-58533
C00662=-85581,-10814,20279,41280,-18093,-59893
C00663=-85551,-10406,21021,40925,-18257,-59713
C00664=-86274,-24518,9978,34497,-20333,-56613
C00665=-91684,-53777,2301,20525,-9313,-33684
C00666=-67305,-55044,34987,1504,5690,-2468
C00667=0,-52280,40443,0,6876,0
C00668=77036,-56616,31288,-2531,4707,4197
C00669=84359,-28321,8817,-32860,-20485,54199
C00670=81156,-16932,14874,-39538,-26422,62851
C00671=93177,-15839,10945,-5896,-17224,48859
C00672=90816,-14121,15571,-13445,-19613,51998
C00673=77970,-27630,4721,-41834,-28549,63607
C00674=81111,-35571,7141,-33980,-21909,52006
C00675=82626,-57814,28323,-4146,3364,6346
C00676=0,-52280,40443,0,6876,0
C00677=0,-28135,76691,0,20839,0
C00678=0,-28135,76691,0,20839,0
C00679=-45332,-39712,59352,-1730,18713,2903
C00680=-94065,-8316,59352,-1730,-37754,-40387
C00681=-100331,-14895,33931,-8215,-36518,-40227
C00682=-98931,-8578,39429,-6260,-48307,-43744
C00683=-100336,-4176,46216,-7600,-55875,-44633
C00684=-93952,8947,73671,995,-68520,-43850
C00685=-98791,-3170,32594,-4861,-60761,-43748
C00686=-98617,4601,38180,-4851,-58752,-43714
C00687=-98986,-12819,-17910,-7864,-33404,-41725
C00688=-98841,-14649,-29255,-9365,-27027,-40913
C00689=-99605,-15546,-21493,-8548,-33053,-41326
C00690=-100467,-8208,-2562,-8095,-44661,-42156
C00691=-98488,7033,71139,-1967,-68237,-42761
C00692=-88754,54,62805,4404,-67858,-45120
C00693=-100222,-4532,45667,-7492,-55263,-44561
C00694=-100331,-14895,33931,-8215,-36518,-40227
C00695=-94065,-8316,59352,-1730,-37754,-40387
C00696=-45544,-32973,71870,-2133,15168,3033
C00697=0,-28135,76691,0,20839,0
C00698=54178,-17846,77779,596,-29686,20997
C00699=54178,-17846,77779,596,-29686,20997
C00700=99462,-18987,75418,611,-28919,20989
C00701=98707,-9390,78674,1080,-71212,38250
C00702=98768,-5182,41096,1808,-44974,38308
C00703=100431,1771,51615,3823,-56746,39115
C00704=97953,-6621,17555,2289,-50176,39420
C00705=95834,-5353,18817,760,-50052,40242
C00706=86453,-3910,18511,-13431,-48443,44868
C00707=88887,-11110,-8515,-11527,-36861,46615
C00708=88808,-13839,-20865,-13699,-30585,47852
C00709=90457,-16080,-12990,-9972,-37305,45724
C00710=97953,-6621,17555,2289,-50176,39420
C00711=100431,1771,51615,3823,-56746,39115
C00712=98768,-5182,41096,1808,-44974,38308
C00713=98707,-9390,78674,1080,-71212,38250
C00714=0,-28135,76691,0,20839,0
C00715=0,-28135,76691,0,20839,0
C00716=-91526,-60598,16699,7584,176,-13289
C00717=-81382,-25890,9219,35455,-25500,-59095
C00718=-81382,-25890,9219,35455,-25500,-59095
C00719=-85509,-13950,19358,32213,-22393,-58041
C00720=-96341,-12683,17919,-5232,-17216,-42057
C00721=-97612,-9184,26280,-8466,-20569,-40722
C00722=-84656,-25369,12054,31249,-26195,-57129
C00723=-82652,-57346,29982,2770,3944,-5064
C00724=0,-52280,40443,0,6876,0
C00725=60653,-54633,35892,-1212,5841,2035
C00726=77942,-28227,6869,-38010,-29303,61907
C00727=82500,-13648,17375,-36975,-24607,62039
C00728=80825,-11424,18929,-41480,-25443,63875
C00729=80510,-10259,22389,-40115,-26795,63066
C00730=64389,-31987,5108,-50419,-37074,66126
C00731=60653,-54633,35892,-1212,5841,2035
C00732=0,-52280,40443,0,6876,0
C00733=0,-28167,76633,0,20843,0
BC00000=413138
BC00001=413138
BC00002=295997
BC00003=264574
BC00004=264574
BC00005=264574
BC00006=264574
BC00007=233852
BC00008=284288
BC00009=284288
BC00010=284288
BC00011=284288
BC00012=284288
BC00013=356545
BC00014=388163
BC00015=356740
BC00016=356740
BC00017=356740
BC00018=356740
BC00019=356740
BC00020=407176
BC00021=407176
BC00022=407176
BC00023=407176
BC00024=407176
BC00025=479433
BC00026=479433
BC00027=479433
BC00028=479433
BC00029=479433
BC00030=530237
BC00031=530237
BC00032=530237
BC00033=530237
BC00034=530237
BC00035=601977
BC00036=601977
BC00037=601977
BC00038=601977
BC00039=601977
BC00040=657723
BC00041=657723
BC00042=657723
BC00043=657723
BC00044=657723
BC00045=601977
BC00046=522422
BC00047=522422
BC00048=671734
BC00049=726463
BC00050=726463
BC00051=726463
BC00052=726463
BC00053=726463
BC00054=782137
BC00055=782137
BC00056=782137
BC00057=782137
BC00058=782137
BC00059=850421
BC00060=850421
BC00061=850421
BC00062=850421
BC00063=850421
BC00064=850421
BC00065=894757
BC00066=894757
BC00067=894757
BC00068=894757
BC00069=894757
BC00070=852119
BC00071=823841
BC00072=755227
BC00073=755227
BC00074=959551
BC00075=959551
BC00076=959551
BC00077=959551
BC00078=959551
BC00079=959551
BC00080=1002575
BC00081=1002575
BC00082=1002575
BC00083=1002575
BC00084=1002575
BC00085=953318
BC00086=927819
BC00087=927819
BC00088=927819
BC00089=943180
BC00090=943180
BC00091=943180
BC00092=943180
BC00093=943180
BC00094=943180
BC00095=943180
BC00096=943180
BC00097=943180
BC00098=943180
BC00099=943180
BC00100=943180
BC00101=943180
BC00102=943180
BC00103=943180
BC00104=943180
BC00105=943180
BC00106=943180
BC00107=943180
BC00108=943180
BC00109=943180
BC00110=943180
BC00111=943180
BC00112=943180
BC00113=943180
BC00114=943182
BC00115=943182
BC00116=943182
BC00117=943182
BC00118=943182
BC00119=943182
BC00120=943182
BC00121=943182
BC00122=943182
BC00123=943182
BC00124=943182
BC00125=943182
BC00126=943182
BC00127=943182
BC00128=943182
BC00129=943182
BC00130=943182
BC00131=943182
BC00132=943182
BC00133=943182
BC00134=943182
BC00135=943182
BC00136=943182
BC00137=943183
BC00138=943184
BC00139=943184
BC00140=943184
BC00141=943184
BC00142=943184
BC00143=943184
BC00144=943184
BC00145=943184
BC00146=943184
BC00147=943184
BC00148=943184
BC00149=943156
BC00150=943170
BC00151=943170
BC00152=943170
BC00153=943170
BC00154=943170
BC00155=943170
BC00156=943170
BC00157=943184
BC00158=943184
BC00159=943184
BC00160=943184
BC00161=943184
BC00162=943184
BC00163=943184
BC00164=943184
BC00165=943184
BC00166=943184
BC00167=943184
BC00168=943184
BC00169=943184
BC00170=943184
BC00171=943184
BC00172=943184
BC00173=943184
BC00174=943184
BC00175=943184
BC00176=943184
BC00177=943184
BC00178=943184
BC00179=943184
BC00180=943184
BC00181=943184
BC00182=911399
BC00183=884954
BC00184=838173
BC00185=838173
BC00186=727925
BC00187=734552
BC00188=750834
BC00189=750837
BC00190=811927
BC00191=811927
BC00192=760768
BC00193=744267
BC00194=744267
BC00195=413138
BC00196=413138
BC00197=413138
BC00198=408626
BC00199=408626
BC00200=408753
BC00201=347392
BC00202=408626
BC00203=408626
BC00204=413138
BC00205=413138
BC00206=413138
BC00207=505502
BC00208=893917
BC00209=915147
BC00210=918406
BC00211=918406
BC00212=918406
BC00213=918406
BC00214=935268
BC00215=935270
BC00216=935270
BC00217=935270
BC00218=935270
BC00219=935270
BC00220=935270
BC00221=935270
BC00222=935270
BC00223=935269
BC00224=935270
BC00225=935271
BC00226=935271
BC00227=935271
BC00228=935271
BC00229=935271
BC00230=935271
BC00231=930781
BC00232=906929
BC00233=936106
BC00234=936109
BC00235=936109
BC00236=936106
BC00237=936107
BC00238=936108
BC00239=936108
BC00240=936109
BC00241=936109
BC00242=936109
BC00243=906929
BC00244=835535
BC00245=835535
BC00246=906929
BC00247=936106
BC00248=936109
BC00249=936109
BC00250=936109
BC00251=936109
BC00252=936114
BC00253=936121
BC00254=936110
BC00255=936109
BC00256=906929
BC00257=835535
BC00258=835535
BC00259=872997
BC00260=918800
BC00261=938197
BC00262=938199
BC00263=938199
BC00264=938199
BC00265=938199
BC00266=938775
BC00267=938199
BC00268=952138
BC00269=952138
BC00270=952138
BC00271=952138
BC00272=952138
BC00273=938197
BC00274=918800
BC00275=872997
BC00276=873283
BC00277=835535
BC00278=872997
BC00279=918800
BC00280=938197
BC00281=938199
BC00282=938199
BC00283=938199
BC00284=938199
BC00285=938199
BC00286=938199
BC00287=938199
BC00288=938199
BC00289=938199
BC00290=938199
BC00291=938197
BC00292=918800
BC00293=849812
BC00294=864290
BC00295=883850
BC00296=922155
BC00297=922155
BC00298=922155
BC00299=922153
BC00300=922155
BC00301=922155
BC00302=922155
BC00303=922153
BC00304=922155
BC00305=914820
BC00306=922155
BC00307=922155
BC00308=922151
BC00309=922153
BC00310=922197
BC00311=922153
BC00312=922155
BC00313=922155
BC00314=922151
BC00315=922153
BC00316=922155
BC00317=922155
BC00318=922155
BC00319=922155
BC00320=918747
BC00321=805523
BC00322=697681
BC00323=697681
BC00324=697681
BC00325=733666
BC00326=758324
BC00327=792433
BC00328=839378
BC00329=839375
BC00330=794510
BC00331=758324
BC00332=697681
BC00333=697681
BC00334=697681
BC00335=841681
BC00336=841681
BC00337=884227
BC00338=901088
BC00339=895224
BC00340=896289
BC00341=925648
BC00342=971783
BC00343=921975
BC00344=907826
BC00345=824879
BC00346=507816
BC00347=507816
BC00348=552804
BC00349=552804
BC00350=551170
BC00351=493239
BC00352=491979
BC00353=285738
BC00354=285865
BC00355=256782
BC00356=258630
BC00357=283526
BC00358=399813
BC00359=552804
BC00360=598286
BC00361=598286
BC00362=616910
BC00363=616910
BC00364=507816
BC00365=507816
BC00366=848972
BC00367=861901
BC00368=977841
BC00369=1011251
BC00370=1011251
BC00371=1011251
BC00372=1011251
BC00373=1011251
BC00374=1018161
BC00375=1018161
BC00376=1018161
BC00377=1018161
BC00378=997427
BC00379=997427
BC00380=997427
BC00381=997427
BC00382=997427
BC00383=997427
BC00384=902188
BC00385=895372
BC00386=895372
BC00387=895372
BC00388=895372
BC00389=895372
BC00390=840744
BC00391=840744
BC00392=840744
BC00393=840744
BC00394=840744
BC00395=840744
BC00396=779300
BC00397=771332
BC00398=771332
BC00399=771332
BC00400=771332
BC00401=771332
BC00402=717855
BC00403=717855
BC00404=717855
BC00405=717855
BC00406=717855
BC00407=717855
BC00408=656405
BC00409=649173
BC00410=649173
BC00411=649173
BC00412=649173
BC00413=649173
BC00414=594961
BC00415=594961
BC00416=594961
BC00417=594961
BC00418=594961
BC00419=594961
BC00420=594961
BC00421=533517
BC00422=525229
BC00423=525229
BC00424=525229
BC00425=525229
BC00426=525229
BC00427=472073
BC00428=472073
BC00429=472073
BC00430=472073
BC00431=472073
BC00432=472073
BC00433=410629
BC00434=405662
BC00435=402968
BC00436=402968
BC00437=402968
BC00438=402968
BC00439=402968
BC00440=402968
BC00441=349186
BC00442=349186
BC00443=349186
BC00444=349186
BC00445=349186
BC00446=349186
BC00447=336469
BC00448=336469
BC00449=336469
BC00450=336469
BC00451=336469
BC00452=336469
BC00453=336469
BC00454=367602
BC00455=367601
BC00456=367601
BC00457=367601
BC00458=367601
BC00459=367601
BC00460=367601
BC00461=425303
BC00462=425303
BC00463=514953
BC00464=463119
BC00465=419862
BC00466=484962
BC00467=484962
BC00468=395463
BC00469=369502
BC00470=369502
BC00471=369502
BC00472=369502
BC00473=369502
BC00474=369502
BC00475=369502
BC00476=369502
BC00477=368885
BC00478=368885
BC00479=368885
BC00480=368885
BC00481=368885
BC00482=368885
BC00483=419064
BC00484=366918
BC00485=349186
BC00486=353241
BC00487=353241
BC00488=353241
BC00489=353241
BC00490=353241
BC00491=410629
BC00492=409135
BC00493=409135
BC00494=409135
BC00495=409135
BC00496=409135
BC00497=472073
BC00498=476126
BC00499=476126
BC00500=476126
BC00501=476126
BC00502=476126
BC00503=533517
BC00504=532644
BC00505=532644
BC00506=532644
BC00507=532644
BC00508=532644
BC00509=594961
BC00510=599988
BC00511=599988
BC00512=599988
BC00513=599988
BC00514=599988
BC00515=656405
BC00516=653254
BC00517=653254
BC00518=653254
BC00519=653254
BC00520=653254
BC00521=717855
BC00522=721570
BC00523=721570
BC00524=721570
BC00525=721570
BC00526=721570
BC00527=779300
BC00528=777963
BC00529=777963
BC00530=777963
BC00531=777963
BC00532=777963
BC00533=840744
BC00534=843810
BC00535=843810
BC00536=843810
BC00537=843810
BC00538=843810
BC00539=902188
BC00540=900128
BC00541=900128
BC00542=900128
BC00543=900128
BC00544=900128
BC00545=998964
BC00546=1000819
BC00547=1000819
BC00548=1000819
BC00549=1000819
BC00550=1000819
BC00551=1000819
BC00552=1000819
BC00553=1000819
BC00554=1000819
BC00555=1000819
BC00556=1000819
BC00557=1000819
BC00558=1000819
BC00559=1000819
BC00560=1000819
BC00561=1000819
BC00562=966834
BC00563=806641
BC00564=769966
BC00565=716686
BC00566=679663
BC00567=721442
BC00568=721442
BC00569=721439
BC00570=781482
BC00571=781888
BC00572=781888
BC00573=781888
BC00574=781888
BC00575=768943
BC00576=718475
BC00577=718475
BC00578=718475
BC00579=778313
BC00580=778313
BC00581=717855
BC00582=792672
BC00583=792672
BC00584=948195
BC00585=948195
BC00586=957587
BC00587=959389
BC00588=1014282
BC00589=1014282
BC00590=1014282
BC00591=1036191
BC00592=1014282
BC00593=978822
BC00594=792672
BC00595=792672
BC00596=792672
BC00597=887446
BC00598=956264
BC00599=956264
BC00600=969252
BC00601=969531
BC00602=1013898
BC00603=1026396
BC00604=982408
BC00605=982408
BC00606=982408
BC00607=956264
BC00608=956264
BC00609=913689
BC00610=792672
BC00611=792672
BC00612=700249
BC00613=546214
BC00614=546214
BC00615=546211
BC00616=546211
BC00617=406776
BC00618=406776
BC00619=352261
BC00620=346119
BC00621=406266
BC00622=406266
BC00623=491556
BC00624=546211
BC00625=546214
BC00626=546214
BC00627=507604
BC00628=410782
BC00629=429690
BC00630=375447
BC00631=350474
BC00632=350474
BC00633=408658
BC00634=408658
BC00635=507604
BC00636=546214
BC00637=546214
BC00638=516757
BC00639=591809
BC00640=591809
BC00641=591809
BC00642=591183
BC00643=650353
BC00644=650538
BC00645=650538
BC00646=584003
BC00647=515801
BC00648=520018
BC00649=520018
BC00650=590597
BC00651=593080
BC00652=593080
BC00653=593081
BC00654=652456
BC00655=652559
BC00656=594501
BC00657=537666
BC00658=433888
BC00659=546211
BC00660=830322
BC00661=830322
BC00662=830322
BC00663=890247
BC00664=890396
BC00665=798848
BC00666=798848
BC00667=798848
BC00668=798848
BC00669=832296
BC00670=845010
BC00671=845010
BC00672=904605
BC00673=904704
BC00674=818840
BC00675=818839
BC00676=818839
BC00677=526967
BC00678=334612
BC00679=334612
BC00680=334612
BC00681=350464
BC00682=350464
BC00683=359337
BC00684=359337
BC00685=359337
BC00686=359337
BC00687=359453
BC00688=359337
BC00689=359337
BC00690=359337
BC00691=359337
BC00692=359337
BC00693=358620
BC00694=350464
BC00695=334612
BC00696=334612
BC00697=334612
BC00698=334613
BC00699=501279
BC00700=501279
BC00701=334612
BC00702=334610
BC00703=349510
BC00704=365935
BC00705=365935
BC00706=365934
BC00707=348430
BC00708=348430
BC00709=348430
BC00710=365935
BC00711=349510
BC00712=334610
BC00713=334612
BC00714=334612
BC00715=512789
BC00716=516757
BC00717=526627
BC00718=466969
BC00719=466969
BC00720=466969
BC00721=523646
BC00722=525745
BC00723=525745
BC00724=525745
BC00725=525745
BC00726=473911
BC00727=473911
BC00728=473911
BC00729=532824
BC00730=533743
BC00731=525745
BC00732=525745
BC00733=525747
///POSTYPE BASE
///RECTAN
///RCONF 0,0,0,0,0,0,0,0,0,0,0,0,0,0,0,0,0,0,0,0,0,0,0,0
P00006=-2.449,0.031,8.825,0.0000,0.0000,0.0000
P00057=0.000,0.000,2.000,0.0000,0.0000,0.0000
P00058=0.000,0.000,3.000,0.0000,0.0000,0.0000
///RCONF 1,0,0,0,0,0,0,0,0,0,0,0,0,0,0,0,0,0,0,0,0,0,0,0
P00097=0.043,-1.896,1.568,0.0000,0.0000,0.0000
P00098=-0.089,-2.467,4.059,0.0000,0.0000,0.0000
P00099=0.011,-2.380,1.226,0.0000,0.0000,0.0000
P00100=-0.081,2.558,4.482,0.0000,0.0000,0.0000
P00101=0.030,-2.286,2.993,0.0000,0.0000,0.0000
P00102=-0.005,-1.108,1.644,0.0000,0.0000,0.0000
P00103=-0.094,-3.400,4.200,0.0000,0.0000,0.0000
P00104=0.043,-2.127,5.826,0.0000,0.0000,0.0000
P00105=-0.043,0.662,5.286,0.0000,0.0000,0.0000
P00106=-0.018,-2.519,0.237,0.0000,0.0000,0.0000
P00107=-0.008,-4.537,-4.500,0.0000,0.0000,0.0000
P00108=0.014,-3.040,2.637,0.0000,0.0000,0.0000
P00109=0.017,-3.622,2.341,0.0000,0.0000,0.0000
P00110=7346.140,158.997,-946.107,-0.1876,37.7131,-155.1643
///RCONF 0,0,0,0,0,0,0,0,0,0,0,0,0,0,0,0,0,0,0,0,0,0,0,0
P00299=-3.815,-1.565,6.918,0.0000,0.0000,0.0000
///RCONF 1,0,0,0,0,0,0,0,0,0,0,0,0,0,0,0,0,0,0,0,0,0,0,0
P00300=-0.036,-1.505,2.318,0.0000,0.0000,0.0000
///RCONF 0,0,0,0,0,0,0,0,0,0,0,0,0,0,0,0,0,0,0,0,0,0,0,0
P00301=0.005,-4.708,-4.628,0.0000,0.0000,0.0000
P00302=0.052,-2.937,-4.426,0.0000,0.0000,0.0000
P00303=-0.004,-1.437,-4.584,0.0000,0.0000,0.0000
P00304=0.028,-1.666,-4.234,0.0000,0.0000,0.0000
P00305=-0.003,-1.920,-3.501,0.0000,0.0000,0.0000
P00306=0.015,-2.252,-3.054,0.0000,0.0000,0.0000
P00307=0.019,-2.151,-5.077,0.0000,0.0000,0.0000
P00308=-0.003,-2.092,-4.888,0.0000,0.0000,0.0000
P00309=-0.040,-2.205,-4.992,0.0000,0.0000,0.0000
P00310=-0.006,-2.490,-5.925,0.0000,0.0000,0.0000
P00311=-0.007,-2.079,-5.307,0.0000,0.0000,0.0000
P00312=-0.032,2.202,-7.632,0.0000,0.0000,0.0000
///RCONF 1,0,0,0,0,0,0,0,0,0,0,0,0,0,0,0,0,0,0,0,0,0,0,0
P00349=0.060,0.167,-1.133,0.0000,0.0000,0.0000
///RCONF 0,0,0,0,0,0,0,0,0,0,0,0,0,0,0,0,0,0,0,0,0,0,0,0
P00350=11.519,-0.008,1.149,0.0000,0.0000,0.0000
P00351=13.563,-0.027,-0.653,0.0000,0.0000,0.0000
P00352=13.252,-0.027,-0.827,0.0000,0.0000,0.0000
P00353=10.971,-0.082,0.776,0.0000,0.0000,0.0000
P00354=-0.024,2.508,-1.824,0.0000,0.0000,0.0000
P00355=-0.001,2.528,-1.131,0.0000,0.0000,0.0000
P00356=-0.034,2.921,-0.262,0.0000,0.0000,0.0000
P00357=0.003,3.386,-0.091,0.0000,0.0000,0.0000
P00358=0.014,3.037,-0.020,0.0000,0.0000,0.0000
P00359=-0.005,2.731,0.912,0.0000,0.0000,0.0000
P00360=-0.011,3.412,0.438,0.0000,0.0000,0.0000
P00361=0.018,3.050,1.253,0.0000,0.0000,0.0000
P00362=0.014,2.784,0.148,0.0000,0.0000,0.0000
P00399=-2.449,0.031,8.825,0.0000,0.0000,0.0000
P00400=5.920,-3.503,-0.024,0.0000,0.0000,0.0000
P00401=3.430,-0.021,1.131,0.0000,0.0000,0.0000
P00402=-0.253,1.107,3.062,0.0000,0.0000,0.0000
P00403=-3.666,-0.015,5.328,0.0000,0.0000,0.0000
P00405=2.420,0.007,1.427,0.0000,0.0000,0.0000
P00406=3.513,-0.022,0.429,0.0000,0.0000,0.0000
P00415=-1.781,-1.303,3.250,0.0000,0.0000,0.0000
P00416=0.027,1.119,3.078,0.0000,0.0000,0.0000
//INST
///DATE 2025/02/25 14:41
///ATTR SC,RW
///GROUP1 RB1,BS1
NOP
CALL JOB:MOVE_INTO_TUNNEL
SFTOF
'------------------------
'------------------------
'SPOINA SRODEK DOL
'------------------------
'------------------------
MOVJ C00000 BC00000 VJ=10.00
MOVJ C00001 BC00001 VJ=30.00
'------------------------
'PODLOGA_BEZ_ROZPORKI
'------------------------
'TEST
MOVL C00002 BC00002 V=166.7
MOVL C00003 BC00003 V=166.7 PL=0
REFP 3 C00004 BC00004
CALL JOB:SEARCH-R1
IMOV P0057 V=23.0
SET P0097 P0006
SFTON P0097
REFP 3 C00005 BC00005
CALL JOB:SEARCH-R1
SET P0097 P0006
SFTON P0097
MOVL C00006 BC00006 V=166.7 PL=0
'TEST
SFTOF
COMM MOVL C00007 BC00007 V=333.3
MOVL C00008 BC00008 V=333.3
'------------------------
'W38 L
'------------------------
'TEST
MOVL C00009 BC00009 V=166.7 PL=0
REFP 3 C00010 BC00010
CALL JOB:SEARCH-R1
IMOV P0057 V=23.0
SET P0098 P0006
SFTON P0098
REFP 3 C00011 BC00011
CALL JOB:SEARCH-R1
SET P0098 P0006
SFTON P0098
MOVL C00012 BC00012 V=166.7 PL=0
'TEST
SFTOF
MOVJ C00013 BC00013 VJ=20.00
'------------------------
'W38 P
'------------------------
'TEST
MOVL C00014 BC00014 V=166.7
MOVL C00015 BC00015 V=166.7 PL=0
REFP 3 C00016 BC00016
CALL JOB:SEARCH-R1
IMOV P0057 V=23.0
SET P0099 P0006
SFTON P0099
REFP 3 C00017 BC00017
CALL JOB:SEARCH-R1
SET P0099 P0006
SFTON P0099
MOVL C00018 BC00018 V=166.7 PL=0
'TEST
SFTOF
MOVL C00019 BC00019 V=333.3
MOVL C00020 BC00020 V=333.3
'------------------------
'W38 L
'------------------------
'TEST
MOVL C00021 BC00021 V=166.7 PL=0
REFP 3 C00022 BC00022
CALL JOB:SEARCH-R1
IMOV P0057 V=23.0
SET P0100 P0006
SFTON P0100
REFP 3 C00023 BC00023
CALL JOB:SEARCH-R1
SET P0100 P0006
SFTON P0100
MOVL C00024 BC00024 V=166.7 PL=0
'TEST
SFTOF
MOVJ C00025 BC00025 VJ=20.00
'------------------------
'W45 P
'------------------------
MOVL C00026 BC00026 V=166.7 PL=0
REFP 3 C00027 BC00027
CALL JOB:SEARCH-R1
IMOV P0057 V=23.0
SET P0101 P0006
SFTON P0101
REFP 3 C00028 BC00028
CALL JOB:SEARCH-R1
SET P0101 P0006
SFTON P0101
MOVL C00029 BC00029 V=166.7 PL=0
'TEST
SFTOF
MOVJ C00030 BC00030 VJ=20.00
'------------------------
'W45 L
'------------------------
MOVL C00031 BC00031 V=133.3 PL=0
REFP 3 C00032 BC00032
CALL JOB:SEARCH-R1
IMOV P0057 V=23.0
SET P0102 P0006
SFTON P0102
REFP 3 C00033 BC00033
CALL JOB:SEARCH-R1
SET P0102 P0006
SFTON P0102
MOVL C00034 BC00034 V=250.0 PL=0
'TEST
SFTOF
MOVJ C00035 BC00035 VJ=20.00
'------------------------
'W48 P
'------------------------
'TEST
MOVL C00036 BC00036 V=133.3 PL=0
REFP 3 C00037 BC00037
CALL JOB:SEARCH-R1
IMOV P0057 V=23.0
SET P0103 P0006
SFTON P0103
REFP 3 C00038 BC00038
CALL JOB:SEARCH-R1
SET P0103 P0006
SFTON P0103
MOVL C00039 BC00039 V=166.7 PL=0
'TEST
SFTOF
MOVL C00040 BC00040 V=416.7
MOVL C00041 BC00041 V=166.7 PL=0
REFP 3 C00042 BC00042
CALL JOB:SEARCH-R1
IMOV P0057 V=23.0
SET P0104 P0006
SFTON P0104
REFP 3 C00043 BC00043
CALL JOB:SEARCH-R1
SET P0104 P0006
SFTON P0104
MOVL C00044 BC00044 V=166.7 PL=0
SFTOF
MOVJ C00045 BC00045 VJ=30.00
MOVJ C00046 BC00046 VJ=30.00
MOVJ C00047 BC00047 VJ=30.00
MOVJ C00048 BC00048 VJ=30.00
MOVJ C00049 BC00049 VJ=20.00
'------------------------
'W36 P
'------------------------
MOVL C00050 BC00050 V=133.3 PL=0
REFP 3 C00051 BC00051
CALL JOB:SEARCH-R1
IMOV P0057 V=23.0
SET P0105 P0006
SFTON P0105
REFP 3 C00052 BC00052
CALL JOB:SEARCH-R1
SET P0105 P0006
SFTON P0105
MOVL C00053 BC00053 V=166.7 PL=0
'TEST
SFTOF
MOVJ C00054 BC00054 VJ=20.00
'------------------------
'W36 L
'------------------------
MOVL C00055 BC00055 V=166.7 PL=0
REFP 3 C00056 BC00056
CALL JOB:SEARCH-R1
IMOV P0057 V=23.0
SET P0106 P0006
SFTON P0106
REFP 3 C00057 BC00057
CALL JOB:SEARCH-R1
SET P0106 P0006
SFTON P0106
MOVL C00058 BC00058 V=166.7 PL=0
'TEST
MOVJ C00059 BC00059 VJ=20.00
SFTOF
'------------------------
'W44 P
'------------------------
'TEST
MOVL C00060 BC00060 V=133.3 PL=0
REFP 3 C00061 BC00061
CALL JOB:SEARCH-R1
IMOV P0057 V=23.0
SET P0107 P0006
SFTON P0107
REFP 3 C00062 BC00062
CALL JOB:SEARCH-R1
SET P0107 P0006
SFTON P0107
MOVL C00063 BC00063 V=250.0 PL=0
'TEST
SFTOF
MOVL C00064 BC00064 V=250.0
MOVL C00065 BC00065 V=333.3
MOVL C00066 BC00066 V=166.7 PL=0
REFP 3 C00067 BC00067
CALL JOB:SEARCH-R1
IMOV P0057 V=23.0
SET P0108 P0006
SFTON P0108
REFP 3 C00068 BC00068
CALL JOB:SEARCH-R1
SET P0108 P0006
SFTON P0108
MOVL C00069 BC00069 V=250.0 PL=0
SFTOF
MOVL C00070 BC00070 V=500.0
MOVJ C00071 BC00071 VJ=25.00
MOVJ C00072 BC00072 VJ=25.00
MOVJ C00073 BC00073 VJ=25.00
MOVJ C00074 BC00074 VJ=30.00
MOVJ C00075 BC00075 VJ=30.00
MOVL C00076 BC00076 V=166.7 PL=0
REFP 3 C00077 BC00077
CALL JOB:SEARCH-R1
IMOV P0057 V=23.0
SET P0109 P0006
SFTON P0109
REFP 3 C00078 BC00078
CALL JOB:SEARCH-R1
SET P0109 P0006
SFTON P0109
MOVL C00079 BC00079 V=250.0 PL=0
'TEST
SFTOF
MOVL C00080 BC00080 V=333.3
MOVL C00081 BC00081 V=166.7 PL=0
REFP 3 C00082 BC00082
CALL JOB:SEARCH-R1
IMOV P0057 V=23.0
SET P0110 P0006
SFTON P0110
REFP 3 C00083 BC00083
CALL JOB:SEARCH-R1
SET P0110 P0006
SFTON P0110
MOVL C00084 BC00084 V=250.0 PL=0
'TEST
SFTOF
MOVL C00085 BC00085 V=250.0
'------------------------
'W44 L
'------------------------
'TEST
CALL JOB:FRONT_SEARCH_0ST-2_5440_V2
COMM MOVJ C00086 BC00086 VJ=20.00
COMM MOVJ C00087 BC00087 VJ=20.00
COMM MOVJ C00088 BC00088 VJ=20.00
COMM 'DODANE
COMM 'SZUKANIE FRONT
COMM '------------------------
COMM '503
COMM '------------------------
COMM MOVL C00089 BC00089 V=333.3
COMM MOVL C00090 BC00090 V=166.7 PL=0
COMM REFP 3 C00091 BC00091
COMM CALL JOB:SEARCH-R1
COMM IMOV P0058 V=16.7
COMM SET P0350 P0006
COMM SFTON P0350
COMM REFP 3 C00092 BC00092
COMM CALL JOB:SEARCH-R1
COMM SET P0350 P0006
COMM SFTON P0350
COMM MOVL C00093 BC00093 V=66.7 PL=0
COMM SFTOF
COMM '------------------------
COMM '------------------------
COMM '502
COMM '------------------------
COMM MOVL C00094 BC00094 V=166.7
COMM MOVL C00095 BC00095 V=66.7 PL=0
COMM REFP 3 C00096 BC00096
COMM CALL JOB:SEARCH-R1
COMM IMOV P0058 V=16.7
COMM SET P0351 P0006
COMM SFTON P0351
COMM REFP 3 C00097 BC00097
COMM CALL JOB:SEARCH-R1
COMM SET P0351 P0006
COMM SFTON P0351
COMM MOVL C00098 BC00098 V=66.7 PL=0
COMM SFTOF
COMM '------------------------
COMM '------------------------
COMM '501
COMM '------------------------
COMM MOVL C00099 BC00099 V=166.7
COMM MOVL C00100 BC00100 V=66.7 PL=0
COMM REFP 3 C00101 BC00101
COMM CALL JOB:SEARCH-R1
COMM IMOV P0058 V=16.7
COMM SET P0352 P0006
COMM SFTON P0352
COMM REFP 3 C00102 BC00102
COMM CALL JOB:SEARCH-R1
COMM SET P0352 P0006
COMM SFTON P0352
COMM MOVL C00103 BC00103 V=66.7 PL=0
COMM SFTOF
COMM '------------------------
COMM '------------------------
COMM '500
COMM '------------------------
COMM MOVL C00104 BC00104 V=166.7
COMM MOVL C00105 BC00105 V=66.7 PL=0
COMM REFP 3 C00106 BC00106
COMM CALL JOB:SEARCH-R1
COMM IMOV P0058 V=16.7
COMM SET P0353 P0006
COMM SFTON P0353
COMM REFP 3 C00107 BC00107
COMM CALL JOB:SEARCH-R1
COMM SET P0353 P0006
COMM SFTON P0353
COMM MOVL C00108 BC00108 V=66.7 PL=0
COMM SFTOF
COMM '------------------------
COMM MOVL C00109 BC00109 V=333.3
COMM MOVL C00110 BC00110 V=333.3
COMM MOVJ C00111 BC00111 VJ=10.00
COMM 'DODANE
COMM MOVJ C00112 BC00112 VJ=10.00
COMM '------------------------
COMM 'SFT402
COMM '------------------------
COMM SFTOF
COMM MOVL C00113 BC00113 V=150.0
COMM MOVL C00114 BC00114 V=66.7 PL=0
COMM REFP 3 C00115 BC00115
COMM CALL JOB:SEARCH-R1
COMM SET P0402 P0006
COMM SFTON P0402
COMM MOVL C00116 BC00116 V=150.0
COMM MOVL C00117 BC00117 V=66.7 PL=0
COMM REFP 3 C00118 BC00118
COMM CALL JOB:SEARCH-R1
COMM SET P0402 P0006
COMM SFTON P0402
COMM MOVL C00119 BC00119 V=133.3
COMM MOVL C00120 BC00120 V=150.0
COMM MOVL C00121 BC00121 V=150.0
COMM MOVL C00122 BC00122 V=66.7 PL=0
COMM REFP 3 C00123 BC00123
COMM CALL JOB:SEARCH-R1
COMM SET P0402 P0006
COMM SFTOF
COMM MOVL C00124 BC00124 V=150.0
COMM '------------------------
COMM 'SFT403
COMM '------------------------
COMM 'START
COMM SFTOF
COMM MOVL C00125 BC00125 V=250.0
COMM MOVL C00126 BC00126 V=133.3 PL=0
COMM REFP 3 C00127 BC00127
COMM CALL JOB:SEARCH-R1
COMM SET P0416 P0006
COMM SFTON P0416
COMM MOVL C00128 BC00128 V=133.3
COMM REFP 3 C00129 BC00129
COMM CALL JOB:SEARCH-R1
COMM SET P0402 P0006
COMM SFTOF
COMM MOVL C00130 BC00130 V=150.0
COMM '------------------------
COMM '------------------------
COMM SFTOF
COMM MOVL C00131 BC00131 V=250.0
COMM MOVL C00132 BC00132 V=133.3 PL=0
COMM REFP 3 C00133 BC00133
COMM CALL JOB:SEARCH-R1
COMM SET P0403 P0006
COMM SFTON P0403
COMM MOVL C00134 BC00134 V=66.7 PL=0
COMM REFP 3 C00135 BC00135
COMM CALL JOB:SEARCH-R1
COMM SET P0403 P0006
COMM SFTOF
COMM MOVL C00136 BC00136 V=150.0
COMM MOVJ C00137 BC00137 VJ=20.00
COMM MOVJ C00138 BC00138 VJ=20.00
COMM '------------------------
COMM 'SFT401
COMM '------------------------
COMM SFTOF
COMM MOVL C00139 BC00139 V=150.0
COMM MOVL C00140 BC00140 V=66.7 PL=0
COMM REFP 3 C00141 BC00141
COMM CALL JOB:SEARCH-R1
COMM SET P0401 P0006
COMM SFTON P0401
COMM MOVL C00142 BC00142 V=66.7 PL=0
COMM REFP 3 C00143 BC00143
COMM CALL JOB:SEARCH-R1
COMM SET P0401 P0006
COMM SFTOF
COMM MOVL C00144 BC00144 V=150.0
COMM 'SFT400
COMM '------------------------
COMM SFTOF
COMM MOVL C00145 BC00145 V=333.3
COMM MOVL C00146 BC00146 V=66.7 PL=0
COMM REFP 3 C00147 BC00147
COMM CALL JOB:SEARCH-R1
COMM SET P0405 P0006
COMM SFTON P0405
COMM MOVL C00148 BC00148 V=66.7 PL=0
COMM REFP 3 C00149 BC00149
COMM CALL JOB:SEARCH-R1
COMM SET P0405 P0006
COMM SFTOF
COMM MOVL C00150 BC00150 V=150.0
COMM 'SFT400
COMM '------------------------
COMM SFTOF
COMM MOVL C00151 BC00151 V=333.3
COMM MOVL C00152 BC00152 V=133.3 PL=0
COMM REFP 3 C00153 BC00153
COMM CALL JOB:SEARCH-R1
COMM SET P0406 P0006
COMM SFTON P0406
COMM MOVL C00154 BC00154 V=66.7 PL=0
COMM REFP 3 C00155 BC00155
COMM CALL JOB:SEARCH-R1
COMM SET P0406 P0006
COMM SFTOF
COMM MOVL C00156 BC00156 V=150.0
COMM 'SFT400
COMM '------------------------
COMM SFTOF
COMM MOVL C00157 BC00157 V=150.0
COMM MOVL C00158 BC00158 V=66.7 PL=0
COMM REFP 3 C00159 BC00159
COMM CALL JOB:SEARCH-R1
COMM SET P0400 P0006
COMM SFTON P0400
COMM MOVL C00160 BC00160 V=150.0
COMM MOVL C00161 BC00161 V=66.7 PL=0
COMM REFP 3 C00162 BC00162
COMM CALL JOB:SEARCH-R1
COMM SET P0400 P0006
COMM SFTON P0400
COMM MOVL C00163 BC00163 V=150.0
COMM MOVL C00164 BC00164 V=150.0
COMM MOVL C00165 BC00165 V=66.7 PL=0
COMM REFP 3 C00166 BC00166
COMM CALL JOB:SEARCH-R1
COMM SET P0400 P0006
COMM SFTOF
COMM MOVL C00167 BC00167 V=83.3
COMM MOVL C00168 BC00168 V=250.0
COMM MOVL C00169 BC00169 V=333.3
COMM MOVL C00170 BC00170 V=66.7 PL=0
COMM REFP 3 C00171 BC00171
COMM CALL JOB:SEARCH-R1
COMM SET P0415 P0006
COMM SFTON P0415
COMM MOVL C00172 BC00172 V=133.3
COMM REFP 3 C00173 BC00173
COMM CALL JOB:SEARCH-R1
COMM SET P0415 P0006
COMM SFTOF
COMM MOVL C00174 BC00174 V=150.0
COMM '------------------------
COMM 'SFT403
COMM '------------------------
COMM 'START
COMM SFTOF
COMM MOVJ C00175 BC00175 VJ=10.00
COMM '------------------------
COMM 'SFT399
COMM '------------------------
COMM 'START
COMM SFTOF
COMM MOVL C00176 BC00176 V=150.0
COMM MOVL C00177 BC00177 V=66.7 PL=0
COMM REFP 3 C00178 BC00178
COMM CALL JOB:SEARCH-R1
COMM SET P0399 P0006
COMM SFTON P0399
COMM MOVL C00179 BC00179 V=66.7 PL=0
COMM REFP 3 C00180 BC00180
COMM CALL JOB:SEARCH-R1
COMM SET P0399 P0006
COMM SFTOF
COMM MOVL C00181 BC00181 V=150.0
COMM MOVJ C00182 BC00182 VJ=20.00
COMM MOVJ C00183 BC00183 VJ=30.00
MOVJ C00184 BC00184 VJ=30.00
MOVJ C00185 BC00185 VJ=30.00
MOVJ C00186 BC00186 VJ=40.00
'WELD
'WELD
MOVJ C00187 BC00187 VJ=20.00
'**********************
'W36
'**********************
MOVL C00188 BC00188 V=500.0
SFTON P0105
MOVL C00189 BC00189 V=166.7 PL=0
SFTOF
MACRO1 MJ#(0) ARGF24
ARCON
SFTON P0106
MOVL C00190 BC00190 V=11.7
ARCOF
SFTOF
MOVJ C00191 BC00191 VJ=15.00
MOVJ C00192 BC00192 VJ=10.00
MOVJ C00193 BC00193 VJ=10.00
MOVJ C00194 BC00194 VJ=20.00
MOVJ C00195 BC00195 VJ=30.00
MOVJ C00196 BC00196 VJ=20.00
MOVJ C00197 BC00197 VJ=10.00
MOVJ C00198 BC00198 VJ=15.00
'**********************
'W38
'**********************
MOVL C00199 BC00199 V=500.0
SFTON P0100
MOVL C00200 BC00200 V=166.7 PL=0
SFTOF
ARCON
SFTON P0099
MOVL C00201 BC00201 V=11.3
ARCOF
SFTOF
'DODANE
MOVL C00202 BC00202 V=500.0
MOVJ C00203 BC00203 VJ=10.00
MOVJ C00204 BC00204 VJ=10.00
MOVJ C00205 BC00205 VJ=10.00
MOVJ C00206 BC00206 VJ=10.00
MOVJ C00207 BC00207 VJ=25.00
COMM '**********************
COMM '**********************
COMM 'POCZATEK SPAWANIA PRZOD
COMM '**********************
COMM '**********************
COMM MOVJ C00208 BC00208 VJ=30.00
COMM MOVL C00209 BC00209 V=416.7
COMM MOVJ C00210 BC00210 VJ=10.00
COMM MOVJ C00211 BC00211 VJ=10.00
COMM MOVL C00212 BC00212 V=150.0
COMM MOVL C00213 BC00213 V=150.0
COMM '**********************
COMM 'W41A SIDE
COMM '**********************
COMM MOVL C00214 BC00214 V=250.0
COMM SFTON P0402
COMM MOVL C00215 BC00215 V=66.7 PL=0
COMM MACRO1 MJ#(0) ARGF14
COMM ARCON
COMM MOVL C00216 BC00216 V=9.2
COMM ARCOF
COMM SFTOF
COMM MOVL C00217 BC00217 V=166.7
COMM '**********************
COMM 'W41A FRONT
COMM '**********************
COMM MOVL C00218 BC00218 V=250.0
COMM SFTON P0350
COMM MOVL C00219 BC00219 V=66.7 PL=0
COMM SFTOF
COMM MACRO1 MJ#(0) ARGF21
COMM ARCON
COMM SFTON P0351
COMM MOVL C00220 BC00220 V=8.3
COMM SFTOF
COMM ARCOF
COMM MOVL C00221 BC00221 V=166.7
COMM '**********************
COMM 'W41B FRONT
COMM '**********************
COMM MOVL C00222 BC00222 V=250.0
COMM SFTON P0352
COMM MOVL C00223 BC00223 V=66.7 PL=0
COMM SFTOF
COMM MACRO1 MJ#(0) ARGF21
COMM ARCON
COMM SFTON P0353
COMM MOVL C00224 BC00224 V=8.3
COMM SFTOF
COMM ARCOF
COMM MOVL C00225 BC00225 V=166.7
COMM MOVL C00226 BC00226 V=100.0
COMM '**********************
COMM 'W41A SIDE
COMM '**********************
COMM SFTON P0400
COMM MOVL C00227 BC00227 V=66.7 PL=0
COMM MACRO1 MJ#(0) ARGF21
COMM ARCON
COMM MOVL C00228 BC00228 V=8.3
COMM ARCOF
COMM SFTOF
COMM MOVL C00229 BC00229 V=166.7
COMM MOVL C00230 BC00230 V=166.7
COMM MOVL C00231 BC00231 V=333.3
COMM MOVJ C00232 BC00232 VJ=20.00
COMM MOVJ C00233 BC00233 VJ=20.00
COMM '**********************
COMM 'W42A.1
COMM '**********************
COMM 'POPRAWIC
COMM MOVL C00234 BC00234 V=500.0
COMM SFTON P0403
COMM MOVL C00235 BC00235 V=66.7 PL=0
COMM MACRO1 MJ#(0) ARGF9
COMM ARCON
COMM MOVL C00236 BC00236 V=9.2
COMM SFTON P0416
COMM MOVL C00237 BC00237 V=9.2
COMM MOVL C00238 BC00238 V=9.2
COMM MOVL C00239 BC00239 V=9.2
COMM SFTON P0402
COMM MOVL C00240 BC00240 V=9.2
COMM MOVL C00241 BC00241 V=9.2
COMM ARCOF
COMM MOVL C00242 BC00242 V=500.0
COMM SFTOF
COMM MOVJ C00243 BC00243 VJ=15.00
COMM 'W42B.1
COMM MOVJ C00244 BC00244 VJ=30.00
COMM MOVJ C00245 BC00245 VJ=30.00
COMM MOVJ C00246 BC00246 VJ=30.00
COMM MOVJ C00247 BC00247 VJ=30.00
COMM '**********************
COMM 'W42B.1
COMM '**********************
COMM MOVL C00248 BC00248 V=500.0
COMM SFTON P0399
COMM MOVL C00249 BC00249 V=66.7 PL=0
COMM MACRO1 MJ#(0) ARGF9
COMM ARCON
COMM SFTON P0415
COMM MOVL C00250 BC00250 V=9.2
COMM MOVL C00251 BC00251 V=9.2
COMM MOVL C00252 BC00252 V=9.2
COMM SFTON P0400
COMM MOVL C00253 BC00253 V=9.2
COMM MOVL C00254 BC00254 V=9.2
COMM ARCOF
COMM MOVL C00255 BC00255 V=500.0
COMM SFTOF
COMM MOVJ C00256 BC00256 VJ=15.00
COMM 'W42A.2
COMM MOVJ C00257 BC00257 VJ=20.00
COMM MOVJ C00258 BC00258 VJ=20.00
COMM MOVJ C00259 BC00259 VJ=20.00
COMM MOVJ C00260 BC00260 VJ=20.00
COMM MOVJ C00261 BC00261 VJ=20.00
COMM '**********************
COMM 'W42A.2
COMM '**********************
COMM MOVL C00262 BC00262 V=500.0
COMM SFTON P0402
COMM MOVL C00263 BC00263 V=66.7 PL=0
COMM SFTOF
COMM MACRO1 MJ#(0) ARGF9
COMM ARCON
COMM SFTON P0402
COMM MOVL C00264 BC00264 V=9.2
COMM ARCOF
COMM MOVL C00265 BC00265 V=166.7
COMM MOVJ C00266 BC00266 VJ=20.00
COMM MOVJ C00267 BC00267 VJ=20.00
COMM MOVL C00268 BC00268 V=166.7
COMM MOVL C00269 BC00269 V=166.7
COMM ARCON
COMM MOVL C00270 BC00270 V=10.8
COMM ARCOF
COMM MOVL C00271 BC00271 V=166.7
COMM MOVJ C00272 BC00272 VJ=10.00
COMM SFTOF
COMM MOVJ C00273 BC00273 VJ=20.00
COMM MOVJ C00274 BC00274 VJ=20.00
COMM MOVJ C00275 BC00275 VJ=20.00
COMM 'W42B.2
COMM MOVJ C00276 BC00276 VJ=20.00
COMM MOVJ C00277 BC00277 VJ=20.00
COMM MOVJ C00278 BC00278 VJ=20.00
COMM MOVJ C00279 BC00279 VJ=20.00
COMM MOVJ C00280 BC00280 VJ=20.00
COMM '**********************
COMM 'W42B.2
COMM '**********************
COMM MOVL C00281 BC00281 V=500.0
COMM SFTON P0400
COMM MOVL C00282 BC00282 V=166.7 PL=0
COMM SFTOF
COMM MACRO1 MJ#(0) ARGF9
COMM ARCON
COMM SFTON P0400
COMM MOVL C00283 BC00283 V=9.2
COMM ARCOF
COMM SFTOF
COMM MOVL C00284 BC00284 V=166.7
COMM MOVL C00285 BC00285 V=166.7
COMM MOVJ C00286 BC00286 VJ=10.00
COMM SFTON P0400
COMM MOVL C00287 BC00287 V=166.7
COMM ARCON
COMM MOVL C00288 BC00288 V=10.8
COMM ARCOF
COMM MOVL C00289 BC00289 V=166.7
COMM MOVL C00290 BC00290 V=500.0
COMM SFTOF
COMM MOVJ C00291 BC00291 VJ=20.00
COMM MOVJ C00292 BC00292 VJ=20.00
COMM 'W42A.3
COMM MOVJ C00293 BC00293 VJ=10.00
COMM MOVJ C00294 BC00294 VJ=20.00
COMM MOVJ C00295 BC00295 VJ=20.00
COMM MOVJ C00296 BC00296 VJ=20.00
COMM '**********************
COMM 'W42A.3
COMM '**********************
COMM MOVL C00297 BC00297 V=500.0
COMM SFTON P0402
COMM MOVL C00298 BC00298 V=166.7 PL=0
COMM MACRO1 MJ#(0) ARGF9
COMM ARCON
COMM MOVL C00299 BC00299 V=9.2
COMM ARCOF
COMM MOVL C00300 BC00300 V=500.0
COMM SFTOF
COMM '**********************
COMM 'W42B.3
COMM '**********************
COMM MOVL C00301 BC00301 V=500.0
COMM SFTON P0400
COMM MOVL C00302 BC00302 V=66.7 PL=0
COMM ARCON
COMM MOVL C00303 BC00303 V=9.2
COMM ARCOF
COMM MOVL C00304 BC00304 V=500.0
COMM SFTOF
COMM MOVJ C00305 BC00305 VJ=10.00
COMM '**********************
COMM 'GORA L
COMM '**********************
COMM MOVL C00306 BC00306 V=500.0
COMM SFTON P0401
COMM MOVL C00307 BC00307 V=66.7 PL=0
COMM MACRO1 MJ#(0) ARGF9
COMM ARCON
COMM MOVL C00308 BC00308 V=11.7
COMM SFTON P0406
COMM MOVL C00309 BC00309 V=11.7
COMM MOVL C00310 BC00310 V=11.7
COMM MOVL C00311 BC00311 V=11.7
COMM ARCOF
COMM MOVL C00312 BC00312 V=500.0
COMM SFTOF
COMM '**********************
COMM 'GORA P
COMM '**********************
COMM MOVL C00313 BC00313 V=166.7
COMM SFTON P0401
COMM MOVL C00314 BC00314 V=166.7 PL=0
COMM ARCON
COMM MOVL C00315 BC00315 V=11.7
COMM SFTON P0405
COMM MOVL C00316 BC00316 V=11.7
COMM MOVL C00317 BC00317 V=11.7
COMM MOVL C00318 BC00318 V=11.7
COMM ARCOF
COMM MOVL C00319 BC00319 V=500.0
COMM SFTOF
COMM MOVJ C00320 BC00320 VJ=10.00
COMM MOVJ C00321 BC00321 VJ=30.00
COMM MOVJ C00322 BC00322 VJ=30.00
COMM 'KONIEC SPAWANIA FRONTU
COMM '**********************
COMM 'W44
COMM '**********************
MOVJ C00323 BC00323 VJ=30.00
MOVJ C00324 BC00324 VJ=30.00
MOVJ C00325 BC00325 VJ=30.00
MOVL C00326 BC00326 V=500.0
SFTON P0107
MOVL C00327 BC00327 V=166.7 PL=0
SFTOF
MACRO1 MJ#(0) ARGF24
ARCON
SFTON P0108
MOVL C00328 BC00328 V=10.8
MOVL C00329 BC00329 V=10.8
ARCOF
SFTOF
MOVL C00330 BC00330 V=500.0
MOVL C00331 BC00331 V=500.0
MOVJ C00332 BC00332 VJ=20.00
MOVJ C00333 BC00333 VJ=20.00
'**********************
'DODATEK
'**********************
MOVJ C00334 BC00334 VJ=10.00
MOVJ C00335 BC00335 VJ=10.00
MOVJ C00336 BC00336 VJ=20.00
MOVJ C00337 BC00337 VJ=20.00
MOVJ C00338 BC00338 VJ=20.00
MOVL C00339 BC00339 V=333.3
MOVL C00340 BC00340 V=166.7
MACRO1 MJ#(0) ARGF24
SFTON P0109
MOVL C00341 BC00341 V=166.7 PL=0
SFTOF
ARCON
SFTON P0108
MOVL C00342 BC00342 V=10.8
ARCOF
SFTOF
MOVL C00343 BC00343 V=500.0
MOVJ C00344 BC00344 VJ=20.00
MOVJ C00345 BC00345 VJ=30.00
'**********************
'W45
'**********************
MOVJ C00346 BC00346 VJ=30.00
MOVJ C00347 BC00347 VJ=20.00
MOVJ C00348 BC00348 VJ=10.00
MACRO1 MJ#(0) ARGF24
MOVL C00349 BC00349 V=500.0
SFTON P0102
MOVL C00350 BC00350 V=166.7 PL=0
SFTOF
ARCON
SFTON P0101
MOVL C00351 BC00351 V=11.7
ARCOF
SFTOF
MOVL C00352 BC00352 V=500.0
'**********************
'SPOINA_PODLOGA_BRAK_ROZP
'**********************
MOVL C00353 BC00353 V=500.0
SFTON P0098
MOVL C00354 BC00354 V=166.7 PL=0
SFTOF
ARCON
SFTON P0097
MOVL C00355 BC00355 V=11.3
ARCOF
SFTOF
'DODANE
MOVL C00356 BC00356 V=500.0
MOVJ C00357 BC00357 VJ=30.00
MOVL C00358 BC00358 V=500.0
MOVJ C00359 BC00359 VJ=30.00
MOVJ C00360 BC00360 VJ=30.00
SFTON P0103
MOVL C00361 BC00361 V=166.7 PL=0
SFTOF
ARCON
SFTON P0104
MOVL C00362 BC00362 V=10.8
ARCOF
SFTOF
MOVL C00363 BC00363 V=500.0
MOVJ C00364 BC00364 VJ=20.00
MOVJ C00365 BC00365 VJ=40.00
CALL JOB:FRONT_WELD_0ST-2_5440_V2
CALL JOB:MOVE_OUT_OF_TUNNEL
CALL JOB:CLEAN-R1
CALL JOB:MOVE_INTO_TUNNEL
MOVJ C00366 BC00366 VJ=30.00 PL=0
'------------------------
'------------------------
'PRAWA STRONA PROFIL GORA
'------------------------
'------------------------
MOVJ C00367 BC00367 VJ=20.00
'------------------------
'W51A L
'------------------------
SFTOF
MOVJ C00368 BC00368 VJ=20.00
MOVL C00369 BC00369 V=333.3 PL=0
REFP 3 C00370 BC00370
CALL JOB:SEARCH-R1
SET P0299 P0006
SFTON P0299
MOVL C00371 BC00371 V=166.7 PL=0
REFP 3 C00372 BC00372
CALL JOB:SEARCH-R1
SET P0299 P0006
SFTON P0299
MOVL C00373 BC00373 V=166.7
MOVL C00374 BC00374 V=333.3
MOVL C00375 BC00375 V=166.7 PL=0
REFP 3 C00376 BC00376
CALL JOB:SEARCH-R1
SET P0299 P0006
SFTON P0299
MOVL C00377 BC00377 V=133.3 PL=0
SFTOF
'------------------------
'W51A P
'------------------------
SFTOF
MOVL C00378 BC00378 V=250.0
MOVL C00379 BC00379 V=66.7 PL=0
REFP 3 C00380 BC00380
CALL JOB:SEARCH-R1
SET P0300 P0006
SFTON P0300
MOVL C00381 BC00381 V=66.7 PL=0
REFP 3 C00382 BC00382
CALL JOB:SEARCH-R1
SET P0300 P0006
SFTON P0300
MOVL C00383 BC00383 V=66.7 PL=0
SFTOF
'------------------------
'W54A L
'------------------------
SFTOF
MOVJ C00384 BC00384 VJ=30.00
MOVL C00385 BC00385 V=133.3 PL=0
REFP 3 C00386 BC00386
CALL JOB:SEARCH-R1
SET P0301 P0006
SFTON P0301
MOVL C00387 BC00387 V=66.7 PL=0
REFP 3 C00388 BC00388
CALL JOB:SEARCH-R1
SET P0301 P0006
SFTON P0301
MOVL C00389 BC00389 V=66.7 PL=0
SFTOF
'------------------------
'W54A P
'------------------------
SFTOF
MOVJ C00390 BC00390 VJ=30.00
MOVL C00391 BC00391 V=133.3 PL=0
REFP 3 C00392 BC00392
CALL JOB:SEARCH-R1
SET P0302 P0006
SFTON P0302
MOVL C00393 BC00393 V=66.7 PL=0
REFP 3 C00394 BC00394
CALL JOB:SEARCH-R1
SET P0302 P0006
SFTON P0302
MOVL C00395 BC00395 V=66.7 PL=0
SFTOF
'------------------------
'W50A L
'------------------------
SFTOF
MOVJ C00396 BC00396 VJ=30.00
MOVL C00397 BC00397 V=133.3 PL=0
REFP 3 C00398 BC00398
CALL JOB:SEARCH-R1
SET P0303 P0006
SFTON P0303
MOVL C00399 BC00399 V=66.7 PL=0
REFP 3 C00400 BC00400
CALL JOB:SEARCH-R1
SET P0303 P0006
SFTON P0303
MOVL C00401 BC00401 V=66.7 PL=0
SFTOF
'------------------------
'W50A P
'------------------------
SFTOF
MOVJ C00402 BC00402 VJ=30.00
MOVL C00403 BC00403 V=133.3 PL=0
REFP 3 C00404 BC00404
CALL JOB:SEARCH-R1
SET P0304 P0006
SFTON P0304
MOVL C00405 BC00405 V=66.7 PL=0
REFP 3 C00406 BC00406
CALL JOB:SEARCH-R1
SET P0304 P0006
SFTON P0304
MOVL C00407 BC00407 V=66.7 PL=0
SFTOF
'------------------------
'W53A L
'------------------------
SFTOF
MOVJ C00408 BC00408 VJ=30.00
MOVL C00409 BC00409 V=133.3 PL=0
REFP 3 C00410 BC00410
CALL JOB:SEARCH-R1
SET P0305 P0006
SFTON P0305
MOVL C00411 BC00411 V=66.7 PL=0
REFP 3 C00412 BC00412
CALL JOB:SEARCH-R1
SET P0305 P0006
SFTON P0305
MOVL C00413 BC00413 V=66.7 PL=0
SFTOF
'------------------------
'W53A P
'------------------------
SFTOF
MOVJ C00414 BC00414 VJ=30.00
MOVL C00415 BC00415 V=200.0
MOVL C00416 BC00416 V=66.7 PL=0
REFP 3 C00417 BC00417
CALL JOB:SEARCH-R1
SET P0306 P0006
SFTON P0306
MOVL C00418 BC00418 V=66.7 PL=0
REFP 3 C00419 BC00419
CALL JOB:SEARCH-R1
SET P0306 P0006
SFTON P0306
MOVL C00420 BC00420 V=66.7 PL=0
SFTOF
'------------------------
'W56A L
'------------------------
SFTOF
MOVJ C00421 BC00421 VJ=30.00
MOVL C00422 BC00422 V=133.3 PL=0
REFP 3 C00423 BC00423
CALL JOB:SEARCH-R1
SET P0307 P0006
SFTON P0307
MOVL C00424 BC00424 V=66.7 PL=0
REFP 3 C00425 BC00425
CALL JOB:SEARCH-R1
SET P0307 P0006
SFTON P0307
MOVL C00426 BC00426 V=66.7 PL=0
SFTOF
'------------------------
'W56A P
'------------------------
SFTOF
MOVJ C00427 BC00427 VJ=30.00
MOVL C00428 BC00428 V=133.3 PL=0
REFP 3 C00429 BC00429
CALL JOB:SEARCH-R1
SET P0308 P0006
SFTON P0308
MOVL C00430 BC00430 V=66.7 PL=0
REFP 3 C00431 BC00431
CALL JOB:SEARCH-R1
SET P0308 P0006
SFTON P0308
MOVL C00432 BC00432 V=66.7 PL=0
SFTOF
'------------------------
'W52A L
'------------------------
SFTOF
MOVJ C00433 BC00433 VJ=30.00
MOVL C00434 BC00434 V=250.0
MOVL C00435 BC00435 V=66.7 PL=0
REFP 3 C00436 BC00436
CALL JOB:SEARCH-R1
SET P0309 P0006
SFTON P0309
MOVL C00437 BC00437 V=66.7 PL=0
REFP 3 C00438 BC00438
CALL JOB:SEARCH-R1
SET P0309 P0006
SFTON P0309
MOVL C00439 BC00439 V=66.7 PL=0
SFTOF
'------------------------
'W52A P
'------------------------
SFTOF
MOVJ C00440 BC00440 VJ=5.00
MOVJ C00441 BC00441 VJ=20.00
MOVL C00442 BC00442 V=116.7 PL=0
REFP 3 C00443 BC00443
CALL JOB:SEARCH-R1
SET P0310 P0006
SFTON P0310
MOVL C00444 BC00444 V=66.7 PL=0
REFP 3 C00445 BC00445
CALL JOB:SEARCH-R1
SET P0310 P0006
SFTON P0310
MOVL C00446 BC00446 V=66.7 PL=0
SFTOF
'------------------------
'W55A L
'------------------------
SFTOF
MOVL C00447 BC00447 V=250.0
MOVJ C00448 BC00448 VJ=10.00
MOVL C00449 BC00449 V=66.7 PL=0
REFP 3 C00450 BC00450
CALL JOB:SEARCH-R1
SET P0311 P0006
SFTON P0311
MOVL C00451 BC00451 V=66.7 PL=0
REFP 3 C00452 BC00452
CALL JOB:SEARCH-R1
SET P0311 P0006
SFTON P0311
MOVL C00453 BC00453 V=66.7 PL=0
SFTOF
'------------------------
'W55A P
'------------------------
SFTOF
MOVL C00454 BC00454 V=250.0
MOVL C00455 BC00455 V=166.7
MOVL C00456 BC00456 V=66.7 PL=0
REFP 3 C00457 BC00457
CALL JOB:SEARCH-R1
SET P0311 P0006
SFTON P0311
MOVL C00458 BC00458 V=66.7 PL=0
REFP 3 C00459 BC00459
CALL JOB:SEARCH-R1
SET P0311 P0006
SFTON P0311
MOVL C00460 BC00460 V=66.7 PL=0
MOVL C00461 BC00461 V=166.7
SFTOF
MOVL C00462 BC00462 V=250.0
MOVJ C00463 BC00463 VJ=20.00
MOVJ C00464 BC00464 VJ=20.00
MOVJ C00465 BC00465 VJ=20.00
MOVJ C00466 BC00466 VJ=20.00
MOVJ C00467 BC00467 VJ=20.00
MOVJ C00468 BC00468 VJ=20.00
'------------------------
'------------------------
'LEWA STRONA PROFIL GORA
'------------------------
'------------------------
MOVJ C00469 BC00469 VJ=10.00
'------------------------
'W55B L
'------------------------
SFTOF
MOVJ C00470 BC00470 VJ=10.00
MOVL C00471 BC00471 V=66.7 PL=0
REFP 3 C00472 BC00472
CALL JOB:SEARCH-R1
SET P0349 P0006
SFTON P0349
MOVL C00473 BC00473 V=66.7 PL=0
REFP 3 C00474 BC00474
CALL JOB:SEARCH-R1
SET P0349 P0006
SFTON P0349
MOVL C00475 BC00475 V=66.7 PL=0
SFTOF
MOVJ C00476 BC00476 VJ=10.00
MOVJ C00477 BC00477 VJ=10.00
'------------------------
'W55B P
'------------------------
SFTOF
MOVL C00478 BC00478 V=66.7 PL=0
REFP 3 C00479 BC00479
CALL JOB:SEARCH-R1
SET P0350 P0006
SFTON P0350
MOVL C00480 BC00480 V=66.7 PL=0
REFP 3 C00481 BC00481
CALL JOB:SEARCH-R1
SET P0350 P0006
SFTON P0350
MOVL C00482 BC00482 V=66.7 PL=0
SFTOF
'------------------------
'W52B L
'------------------------
SFTOF
MOVJ C00483 BC00483 VJ=20.00
MOVJ C00484 BC00484 VJ=20.00
MOVL C00485 BC00485 V=150.0
MOVL C00486 BC00486 V=66.7 PL=0
REFP 3 C00487 BC00487
CALL JOB:SEARCH-R1
SET P0351 P0006
SFTON P0351
MOVL C00488 BC00488 V=66.7 PL=0
REFP 3 C00489 BC00489
CALL JOB:SEARCH-R1
SET P0351 P0006
SFTON P0351
MOVL C00490 BC00490 V=66.7 PL=0
SFTOF
'------------------------
'W52B P
'------------------------
SFTOF
MOVJ C00491 BC00491 VJ=30.00
MOVL C00492 BC00492 V=116.7 PL=0
REFP 3 C00493 BC00493
CALL JOB:SEARCH-R1
SET P0352 P0006
SFTON P0352
MOVL C00494 BC00494 V=66.7 PL=0
REFP 3 C00495 BC00495
CALL JOB:SEARCH-R1
SET P0352 P0006
SFTON P0352
MOVL C00496 BC00496 V=66.7 PL=0
SFTOF
'------------------------
'W56B L
'------------------------
SFTOF
MOVJ C00497 BC00497 VJ=30.00
MOVL C00498 BC00498 V=116.7 PL=0
REFP 3 C00499 BC00499
CALL JOB:SEARCH-R1
SET P0353 P0006
SFTON P0353
MOVL C00500 BC00500 V=66.7 PL=0
REFP 3 C00501 BC00501
CALL JOB:SEARCH-R1
SET P0353 P0006
SFTON P0353
MOVL C00502 BC00502 V=66.7 PL=0
SFTOF
'------------------------
'W56B P
'------------------------
SFTOF
MOVJ C00503 BC00503 VJ=30.00
MOVL C00504 BC00504 V=116.7 PL=0
REFP 3 C00505 BC00505
CALL JOB:SEARCH-R1
SET P0354 P0006
SFTON P0354
MOVL C00506 BC00506 V=66.7 PL=0
REFP 3 C00507 BC00507
CALL JOB:SEARCH-R1
SET P0354 P0006
SFTON P0354
MOVL C00508 BC00508 V=66.7 PL=0
SFTOF
'------------------------
'W53B L
'------------------------
SFTOF
MOVJ C00509 BC00509 VJ=30.00
MOVL C00510 BC00510 V=116.7 PL=0
REFP 3 C00511 BC00511
CALL JOB:SEARCH-R1
SET P0355 P0006
SFTON P0355
MOVL C00512 BC00512 V=66.7 PL=0
REFP 3 C00513 BC00513
CALL JOB:SEARCH-R1
SET P0355 P0006
SFTON P0355
MOVL C00514 BC00514 V=66.7 PL=0
SFTOF
'------------------------
'W53B P
'------------------------
SFTOF
MOVJ C00515 BC00515 VJ=30.00
MOVL C00516 BC00516 V=116.7 PL=0
REFP 3 C00517 BC00517
CALL JOB:SEARCH-R1
SET P0356 P0006
SFTON P0356
MOVL C00518 BC00518 V=66.7 PL=0
REFP 3 C00519 BC00519
CALL JOB:SEARCH-R1
SET P0356 P0006
SFTON P0356
MOVL C00520 BC00520 V=66.7 PL=0
SFTOF
'------------------------
'W50B L
'------------------------
SFTOF
MOVJ C00521 BC00521 VJ=30.00
MOVL C00522 BC00522 V=116.7 PL=0
REFP 3 C00523 BC00523
CALL JOB:SEARCH-R1
SET P0357 P0006
SFTON P0357
MOVL C00524 BC00524 V=66.7 PL=0
REFP 3 C00525 BC00525
CALL JOB:SEARCH-R1
SET P0357 P0006
SFTON P0357
MOVL C00526 BC00526 V=66.7 PL=0
SFTOF
'------------------------
'W50B P
'------------------------
SFTOF
MOVJ C00527 BC00527 VJ=30.00
MOVL C00528 BC00528 V=116.7 PL=0
REFP 3 C00529 BC00529
CALL JOB:SEARCH-R1
SET P0358 P0006
SFTON P0358
MOVL C00530 BC00530 V=66.7 PL=0
REFP 3 C00531 BC00531
CALL JOB:SEARCH-R1
SET P0358 P0006
SFTON P0358
MOVL C00532 BC00532 V=66.7 PL=0
SFTOF
'------------------------
'W54B L
'------------------------
SFTOF
MOVJ C00533 BC00533 VJ=30.00
MOVL C00534 BC00534 V=116.7 PL=0
REFP 3 C00535 BC00535
CALL JOB:SEARCH-R1
SET P0359 P0006
SFTON P0359
MOVL C00536 BC00536 V=66.7 PL=0
REFP 3 C00537 BC00537
CALL JOB:SEARCH-R1
SET P0359 P0006
SFTON P0359
MOVL C00538 BC00538 V=66.7 PL=0
SFTOF
'------------------------
'W54B P
'------------------------
SFTOF
MOVJ C00539 BC00539 VJ=30.00
MOVL C00540 BC00540 V=116.7 PL=0
REFP 3 C00541 BC00541
CALL JOB:SEARCH-R1
SET P0360 P0006
SFTON P0360
MOVL C00542 BC00542 V=66.7 PL=0
REFP 3 C00543 BC00543
CALL JOB:SEARCH-R1
SET P0360 P0006
SFTON P0360
MOVL C00544 BC00544 V=250.0 PL=0
SFTOF
'------------------------
'W51B L
'------------------------
SFTOF
MOVJ C00545 BC00545 VJ=30.00
MOVL C00546 BC00546 V=166.7 PL=0
REFP 3 C00547 BC00547
CALL JOB:SEARCH-R1
SET P0361 P0006
SFTON P0361
MOVL C00548 BC00548 V=66.7 PL=0
REFP 3 C00549 BC00549
CALL JOB:SEARCH-R1
SET P0361 P0006
SFTON P0361
MOVL C00550 BC00550 V=166.7 PL=0
SFTOF
'------------------------
'W51B P
'------------------------
SFTOF
MOVL C00551 BC00551 V=166.7
MOVL C00552 BC00552 V=166.7 PL=0
REFP 3 C00553 BC00553
CALL JOB:SEARCH-R1
SET P0362 P0006
SFTON P0362
MOVL C00554 BC00554 V=66.7 PL=0
REFP 3 C00555 BC00555
CALL JOB:SEARCH-R1
SET P0362 P0006
SFTON P0362
MOVL C00556 BC00556 V=83.3
MOVL C00557 BC00557 V=133.3 PL=0
REFP 3 C00558 BC00558
CALL JOB:SEARCH-R1
SET P0362 P0006
SFTON P0362
SFTOF
MOVL C00559 BC00559 V=250.0
MOVL C00560 BC00560 V=250.0
MOVL C00561 BC00561 V=500.0
MOVJ C00562 BC00562 VJ=20.00
MOVJ C00563 BC00563 VJ=30.00
MOVJ C00564 BC00564 VJ=50.00
MOVJ C00565 BC00565 VJ=40.00
'**********************
'**********************
'POCZATEK SPAWANIA BOKI
'**********************
'**********************
MOVJ C00566 BC00566 VJ=30.00
MOVJ C00567 BC00567 VJ=20.00
'**********************
'W50A
'**********************
MOVL C00568 BC00568 V=250.0
SFTON P0304
MOVL C00569 BC00569 V=166.7 PL=0
SFTOF
MACRO1 MJ#(0) ARGF10
ARCON
SFTON P0303
MOVL C00570 BC00570 V=10.8
ARCOF
SFTOF
MOVL C00571 BC00571 V=250.0
'W13B
MOVJ C00572 BC00572 VJ=20.00
MOVJ C00573 BC00573 VJ=40.00
MOVJ C00574 BC00574 VJ=20.00
MOVJ C00575 BC00575 VJ=20.00
MOVJ C00576 BC00576 VJ=20.00
'**********************
'W50B
'**********************
MOVL C00577 BC00577 V=250.0
SFTON P0357
MOVL C00578 BC00578 V=166.7 PL=0
SFTOF
MACRO1 MJ#(0) ARGF10
ARCON
SFTON P0358
MOVL C00579 BC00579 V=10.8
ARCOF
SFTOF
MOVL C00580 BC00580 V=250.0
MOVJ C00581 BC00581 VJ=50.00
MOVJ C00582 BC00582 VJ=50.00
MOVJ C00583 BC00583 VJ=50.00
MOVJ C00584 BC00584 VJ=50.00
'**********************
'W51A
'**********************
MOVL C00585 BC00585 V=666.7
MOVL C00586 BC00586 V=500.0
SFTON P0300
MOVL C00587 BC00587 V=166.7 PL=0
SFTOF
MACRO1 MJ#(0) ARGF10
ARCON
SFTON P0299
MOVL C00588 BC00588 V=10.8
MOVL C00589 BC00589 V=10.8
ARCOF
MOVL C00590 BC00590 V=166.7
MOVL C00591 BC00591 V=133.3 PL=0
ARCON
MOVL C00592 BC00592 V=8.3
ARCOF
SFTOF
MOVL C00593 BC00593 V=333.3
MOVJ C00594 BC00594 VJ=30.00
MOVJ C00595 BC00595 VJ=50.00
MOVJ C00596 BC00596 VJ=50.00
MOVJ C00597 BC00597 VJ=50.00
MOVJ C00598 BC00598 VJ=30.00
'**********************
'W51B
'**********************
MOVL C00599 BC00599 V=666.7
MOVL C00600 BC00600 V=500.0
SFTON P0361
MOVL C00601 BC00601 V=166.7 PL=0
SFTOF
MACRO1 MJ#(0) ARGF10
ARCON
SFTON P0362
MOVL C00602 BC00602 V=10.8
MOVL C00603 BC00603 V=10.8
ARCOF
MOVL C00604 BC00604 V=166.7
MACRO1 MJ#(0) ARGF9
MOVL C00605 BC00605 V=166.7 PL=0
ARCON
MOVL C00606 BC00606 V=8.3
ARCOF
SFTOF
MOVL C00607 BC00607 V=333.3
MOVL C00608 BC00608 V=250.0
MOVJ C00609 BC00609 VJ=30.00
MOVJ C00610 BC00610 VJ=50.00
MOVJ C00611 BC00611 VJ=50.00
MOVJ C00612 BC00612 VJ=60.00
MOVJ C00613 BC00613 VJ=80.00
MOVJ C00614 BC00614 VJ=40.00
MOVJ C00615 BC00615 VJ=40.00
MOVJ C00616 BC00616 VJ=40.00
MOVJ C00617 BC00617 VJ=30.00
MOVJ C00618 BC00618 VJ=30.00
'**********************
'W52A
'**********************
SFTON P0310
MOVL C00619 BC00619 V=500.0
MOVL C00620 BC00620 V=166.7 PL=0
SFTOF
MACRO1 MJ#(0) ARGF10
ARCON
SFTON P0309
MOVL C00621 BC00621 V=10.8
ARCOF
SFTOF
MOVL C00622 BC00622 V=333.3
MOVJ C00623 BC00623 VJ=50.00
MOVJ C00624 BC00624 VJ=30.00
MOVJ C00625 BC00625 VJ=50.00
MOVJ C00626 BC00626 VJ=50.00
MOVJ C00627 BC00627 VJ=50.00
MOVJ C00628 BC00628 VJ=30.00
MOVJ C00629 BC00629 VJ=20.00
MOVJ C00630 BC00630 VJ=20.00
'**********************
'52B
'**********************
MOVL C00631 BC00631 V=500.0
SFTON P0351
MOVL C00632 BC00632 V=83.3 PL=0
SFTOF
MACRO1 MJ#(0) ARGF10
ARCON
SFTON P0352
MOVL C00633 BC00633 V=10.8
ARCOF
MOVL C00634 BC00634 V=333.3
SFTOF
MOVJ C00635 BC00635 VJ=20.00
MOVJ C00636 BC00636 VJ=50.00
MOVJ C00637 BC00637 VJ=50.00
'**********************
'W53A
'**********************
MOVJ C00638 BC00638 VJ=50.00
MOVJ C00639 BC00639 VJ=50.00
MOVJ C00640 BC00640 VJ=30.00
'**********************
'W53A
'**********************
SFTON P0306
MOVL C00641 BC00641 V=333.3
MOVL C00642 BC00642 V=166.7 PL=0
SFTOF
MACRO1 MJ#(0) ARGF10
ARCON
SFTON P0305
MOVL C00643 BC00643 V=10.8
ARCOF
SFTOF
MOVL C00644 BC00644 V=250.0
MOVJ C00645 BC00645 VJ=30.00
MOVJ C00646 BC00646 VJ=30.00
MOVJ C00647 BC00647 VJ=50.00
MOVJ C00648 BC00648 VJ=50.00
MOVJ C00649 BC00649 VJ=30.00
MOVJ C00650 BC00650 VJ=50.00
MOVL C00651 BC00651 V=500.0
'**********************
'W53B
'**********************
SFTON P0351
MOVL C00652 BC00652 V=250.0
MOVL C00653 BC00653 V=83.3 PL=0
SFTOF
MACRO1 MJ#(0) ARGF10
ARCON
SFTON P0350
MOVL C00654 BC00654 V=10.8
ARCOF
SFTOF
MOVL C00655 BC00655 V=333.3
MOVJ C00656 BC00656 VJ=30.00
MOVJ C00657 BC00657 VJ=50.00
MOVJ C00658 BC00658 VJ=50.00
MOVJ C00659 BC00659 VJ=30.00
MOVJ C00660 BC00660 VJ=30.00
'**********************
'W54A
'**********************
SFTON P0302
MOVL C00661 BC00661 V=250.0
MOVL C00662 BC00662 V=83.3 PL=0
SFTOF
MACRO1 MJ#(0) ARGF10
ARCON
SFTON P0301
MOVL C00663 BC00663 V=10.8
ARCOF
SFTOF
MOVL C00664 BC00664 V=333.3
MOVJ C00665 BC00665 VJ=50.00
MOVJ C00666 BC00666 VJ=30.00
MOVJ C00667 BC00667 VJ=50.00
MOVJ C00668 BC00668 VJ=50.00
MOVJ C00669 BC00669 VJ=50.00
'**********************
'W54B
'**********************
SFTON P0359
MOVL C00670 BC00670 V=250.0
MOVL C00671 BC00671 V=166.7 PL=0
SFTOF
MACRO1 MJ#(0) ARGF10
ARCON
SFTON P0360
MOVL C00672 BC00672 V=10.8
ARCOF
MOVL C00673 BC00673 V=333.3
SFTOF
MOVJ C00674 BC00674 VJ=50.00
MOVJ C00675 BC00675 VJ=30.00
MOVJ C00676 BC00676 VJ=30.00
MOVJ C00677 BC00677 VJ=60.00
MOVJ C00678 BC00678 VJ=40.00
MOVJ C00679 BC00679 VJ=10.00
MOVJ C00680 BC00680 VJ=10.00
MOVJ C00681 BC00681 VJ=10.00
MOVJ C00682 BC00682 VJ=15.00
MOVJ C00683 BC00683 VJ=15.00
MOVJ C00684 BC00684 VJ=15.00
MOVJ C00685 BC00685 VJ=15.00
'**********************
'W55A
'**********************
SFTON P0311
MOVL C00686 BC00686 V=166.7 PL=0
SFTOF
MACRO1 MJ#(0) ARGF10
ARCON
SFTON P0312
MOVL C00687 BC00687 V=10.8
MOVL C00688 BC00688 V=10.8
ARCOF
SFTOF
MOVL C00689 BC00689 V=150.0
MOVJ C00690 BC00690 VJ=10.00
MOVJ C00691 BC00691 VJ=10.00
MOVJ C00692 BC00692 VJ=10.00
MOVJ C00693 BC00693 VJ=10.00
MOVJ C00694 BC00694 VJ=10.00
MOVJ C00695 BC00695 VJ=20.00
MOVJ C00696 BC00696 VJ=30.00
MOVJ C00697 BC00697 VJ=30.00
MOVJ C00698 BC00698 VJ=20.00
MOVJ C00699 BC00699 VJ=30.00
MOVJ C00700 BC00700 VJ=20.00
MOVJ C00701 BC00701 VJ=20.00
MOVJ C00702 BC00702 VJ=30.00
MOVJ C00703 BC00703 VJ=20.00
MOVJ C00704 BC00704 VJ=20.00
'**********************
'W55B
'**********************
SFTON P0350
MOVL C00705 BC00705 V=333.3
MOVL C00706 BC00706 V=166.7 PL=0
SFTOF
MACRO1 MJ#(0) ARGF10
ARCON
SFTON P0349
MOVL C00707 BC00707 V=10.8
MOVL C00708 BC00708 V=10.8
ARCOF
SFTOF
MOVL C00709 BC00709 V=66.7
MOVJ C00710 BC00710 VJ=10.00
MOVJ C00711 BC00711 VJ=20.00
MOVJ C00712 BC00712 VJ=20.00
MOVJ C00713 BC00713 VJ=20.00
MOVJ C00714 BC00714 VJ=30.00
MOVJ C00715 BC00715 VJ=50.00
MOVJ C00716 BC00716 VJ=50.00
MOVJ C00717 BC00717 VJ=40.00
MOVJ C00718 BC00718 VJ=20.00
'**********************
'W56A
'**********************
SFTON P0308
MOVL C00719 BC00719 V=333.3
MOVL C00720 BC00720 V=166.7 PL=0
SFTOF
MACRO1 MJ#(0) ARGF10
ARCON
SFTON P0307
MOVL C00721 BC00721 V=10.8
ARCOF
SFTOF
MOVL C00722 BC00722 V=333.3
MOVJ C00723 BC00723 VJ=50.00
MOVJ C00724 BC00724 VJ=30.00
MOVJ C00725 BC00725 VJ=30.00
MOVJ C00726 BC00726 VJ=30.00
'**********************
'W56B
'**********************
SFTON P0353
MOVL C00727 BC00727 V=250.0
MOVL C00728 BC00728 V=166.7 PL=0
SFTOF
MACRO1 MJ#(0) ARGF10
ARCON
SFTON P0354
MOVL C00729 BC00729 V=10.8
ARCOF
SFTOF
MOVL C00730 BC00730 V=333.3
MOVJ C00731 BC00731 VJ=50.00
MOVJ C00732 BC00732 VJ=50.00
MOVJ C00733 BC00733 VJ=50.00
CALL JOB:MOVE_OUT_OF_TUNNEL
CALL JOB:R1-HOME
END
